// oaksLibrary/Regulatorer/fbSequenceController7Stages
// Pi-regulator 5-sekvens
{attribute 'initialize_on_call'}
FUNCTION_BLOCK fbSequenceController7Stages
VAR_INPUT
	bEnable : BOOL; // Aktiverar reglering
	rProcessValue : REAL; // Aktuellt Ärvärde 
	rSetpoint : REAL; // Aktuellt börvärde. Önskas separat kylbörvärde för kylsekvenser se inputen rCoolSetpoint.
	{attribute 'initialize_on_call'}
	rCoolSetpoint : REFERENCE TO REAL; //Om man önskar ha ett högre börvärde för kylsekvenser lägg denna här så väljs detta på de sekvenser där bActnSequenceX = TRUE. Lämnar man inputen tom körs rSetpoint på både kyl och värmesekvenser.
	rMinSeq1 : REAL := 0; 
	rMaxSeq1 : REAL := 100;
	bActnSequence1 : BOOL; // Gångriktning reglersekvens  (kylsekvens = TRUE)
	bBlockSequence1 : BOOL; // blockera denna sekvens kan användas exempelvis vid nattkyla
	rMinSeq2 : REAL := 0; 
	rMaxSeq2 : REAL := 100;
	bActnSequence2 : BOOL; // Gångriktning reglersekvens  (kylsekvens = TRUE)
	bBlockSequence2 : BOOL; // blockera denna sekvens kan användas exempelvis vid nattkyla
	rMinSeq3 : REAL := 0; 
	rMaxSeq3 : REAL := 100;
	bActnSequence3 : BOOL; // Gångriktning reglersekvens  (kylsekvens = TRUE)
	bBlockSequence3 : BOOL; // blockera denna sekvens kan användas exempelvis vid nattkyla
	rMinSeq4 : REAL := 0; 
	rMaxSeq4 : REAL := 100;
	bActnSequence4 : BOOL; // Gångriktning reglersekvens  (kylsekvens = TRUE)
	bBlockSequence4 : BOOL; // blockera denna sekvens kan användas exempelvis vid nattkyla
	rMinSeq5 : REAL := 0; 
	rMaxSeq5 : REAL := 100;
	bActnSequence5 : BOOL; // Gångriktning reglersekvens  (kylsekvens = TRUE)
	bBlockSequence5 : BOOL; // blockera denna sekvens kan användas exempelvis vid nattkyla
	rMinSeq6 : REAL := 0; 
	rMaxSeq6 : REAL := 100;
	bActnSequence6 : BOOL; // Gångriktning reglersekvens  (kylsekvens = TRUE)
	bBlockSequence6 : BOOL; // blockera denna sekvens kan användas exempelvis vid nattkyla
	rMinSeq7 : REAL := 0; 
	rMaxSeq7 : REAL := 100;
	bActnSequence7 : BOOL; // Gångriktning reglersekvens  (kylsekvens = TRUE)
	bBlockSequence7 : BOOL; // blockera denna sekvens kan användas exempelvis vid nattkyla
	rKpSequence1 : REAL; // Kp
	rKiSequence1 : UDINT; // Ki
	rDiSequence1 : UDINT; // D-tid (Derivata)
	rFDiSequence1 : UDINT; // Filter tid D (Derivata)
	rDzSequence1 : REAL :=0.1; //Dödzon
	rKpSequence2 : REAL; // Kp
	rKiSequence2 : UDINT; // Ki
	rDiSequence2 : UDINT; // D-tid (Derivata)
	rFDiSequence2 : UDINT; // Filter tid D (Derivata)
	rDzSequence2 : REAL :=0.1; //Dödzon
	rKpSequence3 : REAL; // Kp
	rKiSequence3 : UDINT; // Ki
	rDiSequence3 : UDINT; // D-tid (Derivata)
	rFDiSequence3 : UDINT; // Filter tid D (Derivata)
	rDzSequence3 : REAL :=0.1; //Dödzon
	rKpSequence4 : REAL; // Kp
	rKiSequence4 : UDINT; // Ki
	rDiSequence4 : UDINT; // D-tid (Derivata)
	rFDiSequence4 : UDINT; // Filter tid D (Derivata)
	rDzSequence4 : REAL :=0.1; //Dödzon
	rKpSequence5 : REAL; // Kp
	rKiSequence5 : UDINT; // Ki
	rDiSequence5 : UDINT; // D-tid (Derivata)
	rFDiSequence5 : UDINT; // Filter tid D (Derivata)
	rDzSequence5 : REAL :=0.1; //Dödzon
	rKpSequence6 : REAL; // Kp
	rKiSequence6 : UDINT; // Ki
	rDiSequence6 : UDINT; // D-tid (Derivata)
	rFDiSequence6 : UDINT; // Filter tid D (Derivata)
	rDzSequence6 : REAL :=0.1; //Dödzon
	rKpSequence7 : REAL; // Kp
	rKiSequence7 : UDINT; // Ki
	rDiSequence7 : UDINT; // D-tid (Derivata)
	rFDiSequence7 : UDINT; // Filter tid D (Derivata)
	rDzSequence7 : REAL :=0.1; //Dödzon
	iStartSequence : UDINT :=3; //Sekvens där regulator startar
	{attribute 'pingroup' := 'DeviationAlarm'}
	{attribute 'initialize_on_call'}
	rDevLimit : REFERENCE TO REAL := 0;
	{attribute 'pingroup' := 'DeviationAlarm'}
	bBlockHighAlarm : BOOL; // Blockera högtemplarm
	{attribute 'pingroup' := 'DeviationAlarm'}
	bBlockLowAlarm : BOOL; // Blockera lågtemplarm
	{attribute 'pingroup' := 'DeviationAlarm'}
	tAlarmDelay : TIME := T#5S; // larmfördröjning
END_VAR
VAR_OUTPUT
	rY : REAL; // Utsignal huvudregulator
	rOutputSequence1 : REAL;  // regulatorsignal
	rOutputSequence2 : REAL;  // regulatorsignal
	rOutputSequence3 : REAL;  // regulatorsignal
	rOutputSequence4 : REAL;  // regulatorsignal
	rOutputSequence5 : REAL;  // regulatorsignal
	rOutputSequence6 : REAL;  // regulatorsignal
	rOutputSequence7 : REAL;  // regulatorsignal
	{attribute 'pingroup' := 'DeviationAlarm'}
	bAlarmOutput : BOOL; //larmutgång
END_VAR
VAR
	rDevLimitInternal : REAL;
	fbDevAlarmPV: fbDevAlarm;
	rSetPointSequence1,rSetPointSequence2,rSetPointSequence3,rSetPointSequence4,rSetPointSequence5,rSetPointSequence6,rSetPointSequence7 : REAL; 	
	rTempMin,rTempMax : REAL; // tempvariabel för blockering av sekvenser 
	fbSeqLink01: Tc3_BA_Common.FB_BA_SeqLink;
	stSeqLink01 : Tc3_BA_Common.ST_BA_SeqLink;
	fbPidSeq: ARRAY[1..7] OF Tc3_BA_Common.FB_BA_SeqCtrl;
	iStartSequenceInternal : UDINT := 3;
END_VAR

	fbDevAlarmPV(
	tAlarmDelay:=tAlarmDelay , 
	bAutoReset:=TRUE , 
	bAlarmOutput=>bAlarmOutput , 
	bEnable:=bEnable AND mDevAlarmCheck() , 
	rProcessValue:=rProcessValue , 
	rSetPoint:=rSetpoint , 
	rDevLimit:=rDevLimitInternal , 
	bBlockHighAlarm:=bBlockHighAlarm , 
	bBlockLowAlarm:=bBlockLowAlarm );

	IF iStartSequence > 0 AND iStartSequence < 7 THEN
	 iStartSequenceInternal	 := 7 - iStartSequence;
	END_IF;
		
	
	fbSeqLink01(
	bEn:= bEnable, 
	udiSttCtrl:= iStartSequenceInternal, 
	udiIniSwiOvrDly_sec:= 5, 
	rX:= rProcessValue, 
	stSeqLink:=stSeqLink01 , 
	udiCurCtrl=> , 
	bSeqActv=> , 
	bNotRead=> , 
	bNoneOp=> , 
	udiRemTiIniSwiOvrDly_sec=> , 
	bErr=> , 
	sErrDescr=> );
		
	IF bBlockSequence1 THEN
		rTempMin := 0;
		rTempMax := 0;
	ELSE
		rTempMin := rMinSeq1;
		rTempMax := rMaxSeq1;
	END_IF
	rSetPointSequence1 := mCoolSetpointCheck(bActnSequence1);
	fbPidSeq[1](
	bEn:=bEnable , 
	rW:= rSetPointSequence1, 
	rX:=rProcessValue , 
	udiOpMode:= , 
	bActn:=bActnSequence1 , 
	rKp:= rKpSequence1, 
	udiTn_ms:=rKiSequence1*1000 , 
	udiTv_ms:=rDiSequence1*1000 , 
	udiTd_ms:=rFDiSequence1*1000 , 
	rYMax:=rTempMax , 
	rYMin:=rTempMin, 
	rNZ:= rDzSequence1, 
	udiCycCl:= , 
	bSync:= , 
	rSync:= , 
	rYSeqInit:= , 
	udiMyNum:= 7, 
	stSeqLink:=stSeqLink01 , 
	rY=> rOutputSequence1, 
	rE=> , 
	bErr=> , 
	sErrDescr=> );
	
	IF bBlockSequence2 THEN
		rTempMin := 0;
		rTempMax := 0;
	ELSE
		rTempMin := rMinSeq2;
		rTempMax := rMaxSeq2;
	END_IF
	rSetPointSequence2 := mCoolSetpointCheck(bActnSequence2);
	fbPidSeq[2](
	bEn:=bEnable , 
	rW:= rSetPointSequence2, 
	rX:= rProcessValue, 
	udiOpMode:= , 
	bActn:= bActnSequence2, 
	rKp:= rKpSequence2, 
	udiTn_ms:=rKiSequence2*1000 , 
	udiTv_ms:=rDiSequence2*1000 , 
	udiTd_ms:=rFDiSequence2*1000 , 
	rYMax:= rTempMax, 
	rYMin:=rTempMin , 
	rNZ:= rDzSequence2, 
	udiCycCl:= , 
	bSync:= , 
	rSync:= , 
	rYSeqInit:= , 
	udiMyNum:= 6, 
	stSeqLink:= stSeqLink01, 
	rY=> rOutputSequence2, 
	rE=> , 
	bErr=> , 
	sErrDescr=> );
	
	IF bBlockSequence3 THEN
		rTempMin := 0;
		rTempMax := 0;
	ELSE
		rTempMin := rMinSeq3;
		rTempMax := rMaxSeq3;
	END_IF
	rSetPointSequence3 := mCoolSetpointCheck(bActnSequence3);
	fbPidSeq[3](
	bEn:=bEnable , 
	rW:= rSetPointSequence3, 
	rX:= rProcessValue, 
	udiOpMode:= , 
	bActn:= bActnSequence3, 
	rKp:= rKpSequence3, 
	udiTn_ms:=rKiSequence3*1000 , 
	udiTv_ms:=rDiSequence3*1000 , 
	udiTd_ms:=rFDiSequence3*1000 , 
	rYMax:=rTempMax , 
	rYMin:= rTempMin, 
	rNZ:= rDzSequence3, 
	udiCycCl:= , 
	bSync:= , 
	rSync:= , 
	rYSeqInit:= , 
	udiMyNum:= 5, 
	stSeqLink:= stSeqLink01, 
	rY=> rOutputSequence3, 
	rE=> , 
	bErr=> , 
	sErrDescr=> );
	
	IF bBlockSequence4 THEN
		rTempMin := 0;
		rTempMax := 0;
	ELSE
		rTempMin := rMinSeq4;
		rTempMax := rMaxSeq4;
	END_IF
	rSetPointSequence4 := mCoolSetpointCheck(bActnSequence4);
	fbPidSeq[4](
	bEn:=bEnable , 
	rW:= rSetPointSequence4, 
	rX:= rProcessValue, 
	udiOpMode:= , 
	bActn:= bActnSequence4, 
	rKp:= rKpSequence4, 
	udiTn_ms:=rKiSequence4*1000 , 
	udiTv_ms:=rDiSequence4*1000 , 
	udiTd_ms:=rFDiSequence4*1000 , 
	rYMax:=rTempMax , 
	rYMin:= rTempMin, 
	rNZ:= rDzSequence4, 
	udiCycCl:= , 
	bSync:= , 
	rSync:= , 
	rYSeqInit:= , 
	udiMyNum:= 4, 
	stSeqLink:= stSeqLink01, 
	rY=> rOutputSequence4, 
	rE=> , 
	bErr=> , 
	sErrDescr=> );
	
	IF bBlockSequence5 THEN
		rTempMin := 0;
		rTempMax := 0;
	ELSE
		rTempMin := rMinSeq5;
		rTempMax := rMaxSeq5;
	END_IF
	rSetPointSequence5 := mCoolSetpointCheck(bActnSequence5);
	fbPidSeq[5](
	bEn:=bEnable , 
	rW:= rSetPointSequence5, 
	rX:= rProcessValue, 
	udiOpMode:= , 
	bActn:= bActnSequence5, 
	rKp:= rKpSequence5, 
	udiTn_ms:=rKiSequence5*1000 , 
	udiTv_ms:=rDiSequence5*1000 , 
	udiTd_ms:=rFDiSequence5*1000 , 
	rYMax:=rTempMax , 
	rYMin:= rTempMin, 
	rNZ:= rDzSequence5, 
	udiCycCl:= , 
	bSync:= , 
	rSync:= , 
	rYSeqInit:= , 
	udiMyNum:= 3, 
	stSeqLink:= stSeqLink01, 
	rY=> rOutputSequence5, 
	rE=> , 
	bErr=> , 
	sErrDescr=> );
	
	IF bBlockSequence6 THEN
		rTempMin := 0;
		rTempMax := 0;
	ELSE
		rTempMin := rMinSeq6;
		rTempMax := rMaxSeq6;
	END_IF
	rSetPointSequence6 := mCoolSetpointCheck(bActnSequence6);
	fbPidSeq[6](
	bEn:=bEnable , 
	rW:= rSetPointSequence6, 
	rX:= rProcessValue, 
	udiOpMode:= , 
	bActn:= bActnSequence6, 
	rKp:= rKpSequence6, 
	udiTn_ms:=rKiSequence6*1000 , 
	udiTv_ms:=rDiSequence6*1000 , 
	udiTd_ms:=rFDiSequence6*1000 , 
	rYMax:=rTempMax , 
	rYMin:= rTempMin, 
	rNZ:= rDzSequence6, 
	udiCycCl:= , 
	bSync:= , 
	rSync:= , 
	rYSeqInit:= , 
	udiMyNum:= 2, 
	stSeqLink:= stSeqLink01, 
	rY=> rOutputSequence6, 
	rE=> , 
	bErr=> , 
	sErrDescr=> );
	
	IF bBlockSequence7 THEN
		rTempMin := 0;
		rTempMax := 0;
	ELSE
		rTempMin := rMinSeq7;
		rTempMax := rMaxSeq7;
	END_IF
	rSetPointSequence7 := mCoolSetpointCheck(bActnSequence7);
	fbPidSeq[7](
	bEn:=bEnable , 
	rW:= rSetPointSequence7, 
	rX:= rProcessValue, 
	udiOpMode:= , 
	bActn:= bActnSequence7, 
	rKp:= rKpSequence7, 
	udiTn_ms:=rKiSequence7*1000 , 
	udiTv_ms:=rDiSequence7*1000 , 
	udiTd_ms:=rFDiSequence7*1000 , 
	rYMax:=rTempMax , 
	rYMin:= rTempMin, 
	rNZ:= rDzSequence7, 
	udiCycCl:= , 
	bSync:= , 
	rSync:= , 
	rYSeqInit:= , 
	udiMyNum:= 1, 
	stSeqLink:= stSeqLink01, 
	rY=> rOutputSequence7, 
	rE=> , 
	bErr=> , 
	sErrDescr=> );

// Publik metod för att kolla ifall det finns någon kylsekvens i regleringen. Kan exempelvis användas för att blockera högavvikelselarm vid hög utetemperatur då kylsekvens saknas.
METHOD PUBLIC mContainsCoolingSequence : BOOL
mContainsCoolingSequence := bActnSequence1 OR bActnSequence2 OR bActnSequence3 OR bActnSequence4 OR bActnSequence5;
END_METHOD

// Metod för att kolla ifall det är en kylsekvens och om det i sådant fall är något knutet på rCoolSetpoint
METHOD PRIVATE mCoolSetpointCheck : REAL // Valt börvärde
VAR_INPUT
	bActn : BOOL; // Koll av gångriktning
END_VAR
IF NOT bActn THEN
	mCoolSetpointCheck := rSetpoint;
ELSE
	IF __ISVALIDREF(rCoolSetpoint) THEN 
		mCoolSetpointCheck := rCoolSetpoint;
	ELSE
		mCoolSetpointCheck := rSetpoint;
	END_IF
END_IF
END_METHOD

// Kolla ifall något är knutet på inputen rDevLimit. Är inget knutet där inaktiveras avvikelselarmet.
METHOD PRIVATE mDevAlarmCheck : BOOL // Valt börvärde
IF __ISVALIDREF(rDevLimit) THEN 
	mDevAlarmCheck := TRUE;
	rDevLimitInternal := rDevLimit;
ELSE
	mDevAlarmCheck := FALSE;
END_IF
END_METHOD

END_FUNCTION_BLOCK

// oaksLibrary/Skicka värden mellan plc/Inbyggda taggar/fbReadAdsBoolGeneralWp
// Läser önskat real-värde från annan PLC enligt Oaks-standard
// Robert H, 2021-11-23
// Testat 2021-11-23
FUNCTION_BLOCK fbReadAdsBoolGeneralWp
VAR_INPUT
	Enable			: BOOL := TRUE;					// Start
	AmsNetId    	: T_AmsNetId; 					// AMS Net ID till enhet som skall avläsas
    AdsPort     	: T_AmsPort := 851; 			// ADS-port till enhet som skall avläsas
	AdsTimeout    	: TIME := DEFAULT_ADS_TIMEOUT; 	// ADS-timeout
	SymbolName  	: T_MaxString; 					// Symbol-/variabelnamn för den variabel som skall avläsas. Hela sökväg skall anges tex. LA1.GP11.PV
	Interval		: TIME := T#10S;				// Önskat intervall för läsning
	ErrDelay		: TIME := T#5S;					// Larmfördröjning för fel
	FallbackVal		: BOOL;					// Värde vid kom.fel eller manuellt val av fallback (knyt t ex lokal utegivare om den finns)
	UseFallback		: BOOL;							// Sätts om fallbackvärde ska användas automatiskt vid fel
	ForceFallback	: BOOL;							// Sätts om fallbackvärde ska användas ovillkorligt
	Apparatskap 	: STRING := 'ASXX'; 			// Skriv här vilket apparatskåp utetemperaturen tas emot från. Endast för visning i PV4-tagg.
END_VAR
VAR_OUTPUT
	{attribute 'OPC.UA.DA' := '1'}
	Output 			: BOOL; 	//Utetemperatur hämtat från apparatskåp via ADS
	{attribute 'OPC.UA.DA' := '1'}
	FAULT AT %M* 	: BOOL; 	//Kommunikationsfel mottagning av värde via ADS~wp:
	{attribute 'OPC.UA.DA' := '1'}
	PV8 AT %M* 		: STRING;  	//Inställt amsNetId och apparatskåp~wp:
END_VAR
VAR	
	fbReadVal	: fbReadADSBool;
END_VAR

IF Enable THEN
	fbReadVal(enable := Enable, amsNetId := amsNetId, adsPort := adsPort, adsTimeout := adsTimeout, symbolName := SymbolName, interval := interval, errDelay := errDelay, fallbackVal := fallbackVal, useFallback := UseFallback, forceFallback := forceFallback);
	
	Output	:= fbReadVal.bOutputVar;							// Skriv avläst värde					
	PV8		:= CONCAT(amsNetId, CONCAT('-', Apparatskap));		// Bygg ihop ID-sträng för visning
	FAULT	:= fbReadVal.bErr;									// Sätt fellarm
END_IF;

END_FUNCTION_BLOCK

// oaksLibrary/Skicka värden mellan plc/fbReadADSBool
// Läser önskad bool-variabel från annan ADS-enhet
// Robert H, 2021-11-23
// Testat 2021-11-23
FUNCTION_BLOCK fbReadADSBool
VAR_INPUT
    amsNetId    	: T_AmsNetId; 					//AMS Net ID till enhet som skall avläsas
    adsPort     	: T_AmsPort := 851; 			// ADS-port till den enhet som skall avlä
	symbolName  	: T_MaxString; 					// Symbol-/variabelnamn för den variabel som skall avläsas. Hela sökväg skall anges tex. LA1.GP11.PV
	enable			: BOOL;							// Start
	adsTimeout    	: TIME := DEFAULT_ADS_TIMEOUT; 	// ADS-timout
	interval		: TIME := T#10S;				// Önskat intervall för läsning
	errDelay		: TIME := T#5S;					// Larmfördröjning för fel
	fallbackVal		: BOOL := FALSE;				// Värde vid kom.fel eller manuellt val av fallback
	useFallback		: BOOL := FALSE;				// Sätts om fallbackvärde får användas vid fel
	forceFallback	: BOOL := FALSE;				// Sätts om fallbackvärde ska användas ovillkorligt 			
END_VAR
VAR_OUTPUT
	bBusy     	: BOOL; 			// Upptagen
	bErr     	: BOOL; 			// Fel (via Err-flagga från funktioner, eller om case landat i error state över 10 ggr)
	nErrId    	: UDINT;			// Felkod
	SymInfo  	: SYMINFOSTRUCT; 	// Datastruktur avläst symbolinfo
	bOutputVar	: BOOL;				// Avläst värde
END_VAR
VAR
    errInternal   		: BOOL; 					// Fel
	fbErrorTon 			: TON;  					// Tillslagsfördröjning felindikering
	fbErrorTof 			: TOF;						// Frånslagsfördröjning felindikering
	fbReadSymInfoByName	: PLC_ReadSymInfoByName;	// Maska ut symboladress
 	fbAdsRead			: ADSREAD;					// ADS-block 
	state 				: INT;						// Case-index
	CycleTimer			: TON;						// Intervalltimer för ADS-funktioner
	outputValInternal	: BOOL;						// Avläst värde internt
	StErrCnt			: INT;						// Antal gånger i rad case landat i error state
END_VAR

// Från/tillslagsfördröjning kom.fel
fbErrorTof(IN := , PT := interval + T#5S , Q => errInternal);
fbErrorTon(IN := errInternal OR (amsNetId = '') OR (StErrCnt > 10), PT := errDelay);

bErr := fbErrorTon.Q OR amsNetId = '';

CycleTimer(IN := state = 0 AND (NOT bBusy), PT := Interval);	// Intervalltimer för ADS-funktioner

CASE state OF
	0:
		IF CycleTimer.Q AND enable THEN
			bBusy := TRUE;
			fbErrorTof.IN := FALSE;			
			state := 1;
		END_IF	
	
	1: // Read symbol info by specified name
					
			bBusy := TRUE;
			fbErrorTof.IN := FALSE;
					
			fbReadSymInfoByName(
			NETID:= amsNetId, 
			PORT:= adsPort, 
			SYMNAME:= symbolName, 
			START:= TRUE, 
			TMOUT:= adsTimeout, 
			BUSY=> bBusy, 
			ERR=> fbErrorTof.IN, 
			ERRID=> nErrId, 
			SYMINFO=> SymInfo);
			
			IF NOT bBusy THEN
				IF NOT errInternal AND SymInfo.symDataType = 'BOOL' THEN
					fbReadSymInfoByName( Start := FALSE );
					 state := 2; // Success / Goto next
				ELSE
					fbReadSymInfoByName( Start := FALSE );
					state := 100; // Error
				END_IF
			END_IF
		
	2: // Read symbol value
			
			fbAdsRead(
			NETID:= amsNetId, 
			PORT:= adsPort, 
			IDXGRP:= syminfo.idxGroup, 
			IDXOFFS:= syminfo.idxOffset, 
			LEN:= SIZEOF(outputValInternal), 
			DESTADDR:= ADR(outputValInternal), 
			READ:= TRUE, 
			TMOUT:= adsTimeout, 
			BUSY=> bBusy, 
			ERR=> fbErrorTof.IN, 
			ERRID=> nErrId);
									
			IF NOT bBusy THEN
				IF NOT errInternal THEN
					fbAdsRead( READ := FALSE );
					state := 0; // Success / Goto next
					StErrCnt := 0;
				ELSE
					fbAdsRead( READ := FALSE );
					state := 100; // Error
				END_IF
			END_IF
	
	100: // Error handling
	StErrCnt := StErrCnt + 1;	
	state := 0;
END_CASE

IF (bErr AND useFallback) OR forceFallback THEN
	bOutputVar := fallbackVal;
ELSIF bErr THEN
	bOutputVar := FALSE;
ELSE
	bOutputVar := outputValInternal;
END_IF

END_FUNCTION_BLOCK

// oaksLibrary/Skicka värden mellan plc/Inbyggda taggar/fbReadAdsRealGeneralWp
// Läser önskat real-värde från annan PLC enligt Oaks-standard
// Robert H, 2021-11-23
// Testat 2021-11-23
FUNCTION_BLOCK fbReadAdsRealGeneralWp
VAR_INPUT
	Enable			: BOOL := TRUE;					// Start
	AmsNetId    	: T_AmsNetId; 					// AMS Net ID till enhet som skall avläsas
    AdsPort     	: T_AmsPort := 851; 			// ADS-port till enhet som skall avläsas
	AdsTimeout    	: TIME := DEFAULT_ADS_TIMEOUT; 	// ADS-timeout
	SymbolName  	: T_MaxString; 					// Symbol-/variabelnamn för den variabel som skall avläsas. Hela sökväg skall anges tex. LA1.GP11.PV
	Interval		: TIME := T#10S;				// Önskat intervall för läsning
	ErrDelay		: TIME := T#5S;					// Larmfördröjning för fel
	FallbackVal		: REAL := 0.0;					// Värde vid kom.fel eller manuellt val av fallback (knyt t ex lokal utegivare om den finns)
	UseFallback		: BOOL;							// Sätts om fallbackvärde ska användas automatiskt vid fel
	ForceFallback	: BOOL;							// Sätts om fallbackvärde ska användas ovillkorligt
	Apparatskap 	: STRING := 'ASXX'; 			// Skriv här vilket apparatskåp utetemperaturen tas emot från. Endast för visning i PV4-tagg.
END_VAR
VAR_OUTPUT
	{attribute 'OPC.UA.DA' := '1'}
	Output 			: REAL; 	//Värde hämtat från apparatskåp via ADS (Knyts till egenskapad tagg)
	{attribute 'OPC.UA.DA' := '1'}
	FAULT AT %M* 	: BOOL; 	//Kommunikationsfel mottagning av värde via ADS~wp:
	{attribute 'OPC.UA.DA' := '1'}
	PV8 AT %M* 		: STRING;  	//Inställt amsNetId och apparatskåp~wp:
END_VAR
VAR	
	fbReadVal	: fbReadADSReal;
END_VAR

IF Enable THEN
	fbReadVal(enable := Enable, amsNetId := amsNetId, adsPort := adsPort, adsTimeout := adsTimeout, symbolName := SymbolName, interval := interval, errDelay := errDelay, fallbackVal := fallbackVal, useFallback := UseFallback, forceFallback := forceFallback);
	
	Output	:= fbReadVal.rOutputVar;							// Skriv avläst värde					
	PV8		:= CONCAT(amsNetId, CONCAT('-', Apparatskap));		// Bygg ihop ID-sträng för visning
	FAULT	:= fbReadVal.bErr;									// Sätt fellarm
END_IF;

END_FUNCTION_BLOCK

// oaksLibrary/Skicka värden mellan plc/fbReadADSReal
// Läser önskad real-variabel från annan ADS-enhet
// Robert H, 2021-11-23
// Testat 2021-11-23
FUNCTION_BLOCK fbReadADSReal
VAR_INPUT
    amsNetId    	: T_AmsNetId; 					//AMS Net ID till enhet som skall avläsas
    adsPort     	: T_AmsPort := 851; 			// ADS-port till den enhet som skall avlä
	symbolName  	: T_MaxString; 					// Symbol-/variabelnamn för den variabel som skall avläsas. Hela sökväg skall anges tex. LA1.GP11.PV
	enable			: BOOL;							// Start
	adsTimeout    	: TIME := DEFAULT_ADS_TIMEOUT; 	// ADS-timout
	interval		: TIME := T#10S;				// Önskat intervall för läsning
	errDelay		: TIME := T#5S;					// Larmfördröjning för fel
	fallbackVal		: REAL := 0.0;					// Värde vid kom.fel eller manuellt val av fallback
	useFallback		: BOOL := FALSE;				// Sätts om fallbackvärde får användas vid fel
	forceFallback	: BOOL := FALSE;				// Sätts om fallbackvärde ska användas ovillkorligt 			
END_VAR
VAR_OUTPUT
	bBusy     	: BOOL; 			// Upptagen
	bErr     	: BOOL; 			// Fel (via Err-flagga från funktioner, eller om case landat i error state över 10 ggr)
	nErrId    	: UDINT;			// Felkod
	SymInfo  	: SYMINFOSTRUCT; 	// Datastruktur avläst symbolinfo
	rOutputVar	: REAL;				// Avläst värde
END_VAR
VAR
    errInternal   		: BOOL; 					// Fel
	fbErrorTon 			: TON;  					// Tillslagsfördröjning felindikering
	fbErrorTof 			: TOF;						// Frånslagsfördröjning felindikering
	fbReadSymInfoByName	: PLC_ReadSymInfoByName;	// Maska ut symboladress
 	fbAdsRead			: ADSREAD;					// ADS-block 
	state 				: INT;						// Case-index
	CycleTimer			: TON;						// Intervalltimer för ADS-funktioner
	outputValInternal	: REAL;						// Avläst värde internt
	StErrCnt			: INT;						// Antal gånger i rad case landat i error state
END_VAR

// Från/tillslagsfördröjning kom.fel
fbErrorTof(IN := , PT := interval + T#5S , Q => errInternal);
fbErrorTon(IN := errInternal OR (amsNetId = '') OR (StErrCnt > 10), PT := errDelay);

bErr := fbErrorTon.Q OR amsNetId = '';

CycleTimer(IN := state = 0 AND (NOT bBusy), PT := Interval);	// Intervalltimer för ADS-funktioner

CASE state OF
	0:
		IF CycleTimer.Q AND enable THEN
			bBusy := TRUE;
			fbErrorTof.IN := FALSE;			
			state := 1;
		END_IF	
	
	1: // Read symbol info by specified name
					
			bBusy := TRUE;
			fbErrorTof.IN := FALSE;
					
			fbReadSymInfoByName(
			NETID:= amsNetId, 
			PORT:= adsPort, 
			SYMNAME:= symbolName, 
			START:= TRUE, 
			TMOUT:= adsTimeout, 
			BUSY=> bBusy, 
			ERR=> fbErrorTof.IN, 
			ERRID=> nErrId, 
			SYMINFO=> SymInfo);
			
			IF NOT bBusy THEN
				IF NOT errInternal AND SymInfo.symDataType = 'REAL' THEN
					fbReadSymInfoByName( Start := FALSE );
					 state := 2; // Success / Goto next
				ELSE
					fbReadSymInfoByName( Start := FALSE );
					state := 100; // Error
				END_IF
			END_IF
		
	2: // Read symbol value
	
			fbAdsRead(
			NETID:= amsNetId, 
			PORT:= adsPort, 
			IDXGRP:= syminfo.idxGroup, 
			IDXOFFS:= syminfo.idxOffset, 
			LEN:= SIZEOF(outputValInternal), 
			DESTADDR:= ADR(outputValInternal), 
			READ:= TRUE, 
			TMOUT:= adsTimeout, 
			BUSY=> bBusy, 
			ERR=> fbErrorTof.IN, 
			ERRID=> nErrId);
									
			IF NOT bBusy THEN
				IF NOT errInternal THEN
					fbAdsRead( READ := FALSE );
					state := 0; // Success / Goto next
					StErrCnt := 0;
				ELSE
					fbAdsRead( READ := FALSE );
					state := 100; // Error
				END_IF
			END_IF
	
	100: // Error handling
		StErrCnt := StErrCnt + 1;
		state := 0;
END_CASE

IF (bErr AND useFallback) OR forceFallback THEN
	rOutputVar := fallbackVal;
ELSIF bErr THEN
	rOutputVar := 0.0;
ELSE
	rOutputVar := outputValInternal;
END_IF

END_FUNCTION_BLOCK

// oaksLibrary/Skicka värden mellan plc/Inbyggda taggar/fbReadAdsRealOutdoorMeantempWp
// Läser momentan och medelvärde utetemp från annan PLC enligt oaks-standard
// Robert H, 2021-11-23
// Testat 2021-11-23
FUNCTION_BLOCK fbReadAdsRealOutdoorMeantempWp
VAR_INPUT
	Enable			: BOOL := TRUE;					// Start
	AmsNetId    	: T_AmsNetId; 					// AMS Net ID till enhet som skall avläsas
	sApparatskap 	: STRING 	:= 'ASXX'; 			// Skriv här vilket apparatskåp utetemperaturen tas emot från. Endast för visning i PV4-tagg.
    AdsPort     	: T_AmsPort := 851; 			// ADS-port till den enhet som skall avläsas
	AdsTimeout    	: TIME := DEFAULT_ADS_TIMEOUT; 	// ADS-timout
	Interval		: TIME := T#10S;				// Önskat intervall för läsning
	ErrDelay		: TIME := T#5S;					// Larmfördröjning för fel
	UseFallback		: BOOL;							// Sätts om fallbackvärde ska användas automatiskt vid fel
	FallbackVal		: REAL := 0.0;					// Värde vid kom.fel eller manuellt val av fallback (knyt t ex lokal utegivare om den finns)
	ForceFallback	: BOOL;							// Sätts om fallbackvärde ska användas ovillkorligt
END_VAR
VAR_OUTPUT
	{attribute 'OPC.UA.DA' := '1'}
	PV  AT %M* : REAL; //Utetemperatur hämtat från apparatskåp via ads.~wp:[unit]°C[format]0.0
	{attribute 'OPC.UA.DA' := '1'}
	PV1  AT %M* : REAL; //Utetemperatur medel hämtat från apparatskåp via ads.~wp:[unit]°C[format]0.0
	{attribute 'OPC.UA.DA' := '1'}
	FAULT AT %M* : BOOL; //Kommunikationsfel mottagning utetemperatur~wp:
	{attribute 'OPC.UA.DA' := '1'}
	PV4 AT %M* : STRING;   //Inställt amsNetId och apparatskåp~wp:
END_VAR
VAR	
	fbUtetempMom	: fbReadADSReal;
	fbUtetempMed	: fbReadADSReal;
END_VAR

IF enable THEN
	fbUtetempMom(Enable := enable, amsNetId := amsNetId, adsPort := adsPort, adsTimeout := adsTimeout, symbolName := 'oaksGVL.rOutdoorTemp', interval := interval, errDelay := errDelay, fallbackVal := fallbackVal, useFallback := UseFallback, forceFallback := forceFallback);
	oaksGVL.rOutdoorTemp := fbUtetempMom.rOutputVar;
	
	fbUtetempMed(Enable := enable, amsNetId := amsNetId, adsPort := adsPort, adsTimeout := adsTimeout, symbolName := 'oaksGVL.rOutdoorTempMean', interval := interval, errDelay := errDelay, fallbackVal := fallbackVal, useFallback := UseFallback, forceFallback := forceFallback);
	oaksGVL.rOutdoorTempMean := fbUtetempMed.rOutputVar;
	
	PV		:= oaksGVL.rOutdoorTemp;							// Skriv utetemp till utvariabel	
	PV1		:= oaksGVL.rOutdoorTempMean;						// Skriv utetemp medel till utvariabel				
	PV4		:= CONCAT(amsNetId, CONCAT('-', sApparatskap));		// Bygg ihop ID-sträng för visning
	FAULT	:= fbUtetempMom.bErr OR fbUtetempMed.bErr;			// Sätt fel
END_IF;

END_FUNCTION_BLOCK

// oaksLibrary/Skicka värden mellan plc/Inbyggda taggar/fbReadAdsRealOutdoortempWp
// Läser utetemp från annan PLC enligt oaks-standard
// Robert H, 2021-11-23
// Testat 2021-11-23
FUNCTION_BLOCK fbReadAdsRealOutdoortempWp
VAR_INPUT
	Enable			: BOOL := TRUE;					// Start
	AmsNetId    	: T_AmsNetId; 					// AMS Net ID till enhet som skall avläsas
	sApparatskap 	: STRING 	:= 'ASXX'; 			// Skriv här vilket apparatskåp utetemperaturen tas emot från. Endast för visning i PV4-tagg.
    AdsPort     	: T_AmsPort := 851; 			// ADS-port till den enhet som skall avläsas
	AdsTimeout    	: TIME := DEFAULT_ADS_TIMEOUT; 	// ADS-timout
	Interval		: TIME := T#10S;				// Önskat intervall för läsning
	ErrDelay		: TIME := T#5S;					// Larmfördröjning för fel
	UseFallback		: BOOL;							// Sätts om fallbackvärde ska användas automatiskt vid fel
	FallbackVal		: REAL := 0.0;					// Värde vid kom.fel eller manuellt val av fallback (knyt t ex lokal utegivare om den finns)
	ForceFallback	: BOOL;							// Sätts om fallbackvärde ska användas ovillkorligt
END_VAR
VAR_OUTPUT
	{attribute 'OPC.UA.DA' := '1'}
	PV  AT %M* : REAL; //Utetemperatur hämtat från apparatskåp via ads.~wp:[unit]°C[format]0.0
	{attribute 'OPC.UA.DA' := '1'}
	FAULT AT %M* : BOOL; //Kommunikationsfel mottagning utetemperatur~wp:
	{attribute 'OPC.UA.DA' := '1'}
	PV4 AT %M* : STRING;   //Inställt amsNetId och apparatskåp~wp:
END_VAR
VAR	
	fbUtetempMom	: fbReadADSReal;
	fbUtetempMed	: fbReadADSReal;
END_VAR

IF enable THEN
	fbUtetempMom(Enable := enable, amsNetId := amsNetId, adsPort := adsPort, adsTimeout := adsTimeout, symbolName := 'oaksGVL.rOutdoorTemp', interval := interval, errDelay := errDelay, fallbackVal := fallbackVal, useFallback := UseFallback, forceFallback := forceFallback);
	oaksGVL.rOutdoorTemp := fbUtetempMom.rOutputVar;
	
	PV		:= oaksGVL.rOutdoorTemp;							// Skriv utetemp till utvariabel					
	PV4		:= CONCAT(amsNetId, CONCAT('-', sApparatskap));		// Bygg ihop ID-sträng för visning
	FAULT	:= fbUtetempMom.bErr OR fbUtetempMed.bErr;			// Sätt fel
END_IF;

END_FUNCTION_BLOCK

// oaksLibrary/Skicka värden mellan plc/Inbyggda taggar/fbReadAdsTempSensorWp
// Läser tempgivare från annan PLC enligt oaks-standard
// Robert H, 2021-11-23
// Testat 2021-11-23
FUNCTION_BLOCK fbReadAdsTempSensorWp
VAR_INPUT
	Enable			: BOOL := TRUE;					// Start
	AmsNetId    	: T_AmsNetId; 					// AMS Net ID till enhet som skall avläsas
    AdsPort     	: T_AmsPort := 851; 			// ADS-port till enhet som skall avläsas
	AdsTimeout    	: TIME := DEFAULT_ADS_TIMEOUT; 	// ADS-timeout
	SymbolName  	: T_MaxString; 					// Symbol-/variabelnamn för den variabel som skall avläsas. Hela sökväg skall anges tex. LA1.GT11.PV
	Interval		: TIME := T#10S;				// Önskat intervall för läsning
	ErrDelay		: TIME := T#5S;					// Larmfördröjning för fel
	FallbackVal		: REAL := 0.0;					// Värde vid kom.fel eller manuellt val av fallback (knyt t ex lokal utegivare om den finns)
	UseFallback		: BOOL;							// Sätts om fallbackvärde ska användas automatiskt vid fel
	ForceFallback	: BOOL;							// Sätts om fallbackvärde ska användas ovillkorligt
	Apparatskap 	: STRING := 'ASXX'; 			// Skriv här vilket apparatskåp utetemperaturen tas emot från. Endast för visning i PV4-tagg.
END_VAR
VAR_OUTPUT
	{attribute 'OPC.UA.DA' := '1'}
	PV AT %M*		: REAL; 	//Temperatur~wp:[unit]°C[format]0.0[trendoptions]i:300
	{attribute 'OPC.UA.DA' := '1'}
	FAULT AT %M* 	: BOOL; 	//Kommunikationsfel mottagning av värde via ADS~wp:
	{attribute 'OPC.UA.DA' := '1'}
	PV8 AT %M* 		: STRING;  	//Inställt amsNetId och apparatskåp~wp:
END_VAR
VAR	
	fbReadVal	: fbReadADSReal;
END_VAR

IF Enable THEN
	fbReadVal(enable := Enable, amsNetId := amsNetId, adsPort := adsPort, adsTimeout := adsTimeout, symbolName := SymbolName, interval := interval, errDelay := errDelay, fallbackVal := fallbackVal, useFallback := UseFallback, forceFallback := forceFallback);
	
	PV		:= fbReadVal.rOutputVar;							// Skriv avläst värde					
	PV8		:= CONCAT(amsNetId, CONCAT('-', Apparatskap));		// Bygg ihop ID-sträng för visning
	FAULT	:= fbReadVal.bErr;									// Sätt fellarm
END_IF;

END_FUNCTION_BLOCK

// oaksLibrary/Skicka värden mellan plc/fbReadAdsInt
// Läser önskad int-variabel från annan ADS-enhet
// Robert H, 2021-11-23
// Testat 2021-11-23
FUNCTION_BLOCK fbReadAdsInt
VAR_INPUT
    amsNetId    	: T_AmsNetId; 					//AMS Net ID till enhet som skall avläsas
    adsPort     	: T_AmsPort := 851; 			// ADS-port till den enhet som skall avlä
	symbolName  	: T_MaxString; 					// Symbol-/variabelnamn för den variabel som skall avläsas. Hela sökväg skall anges tex. LA1.GP11.PV
	enable			: BOOL;							// Start
	adsTimeout    	: TIME := DEFAULT_ADS_TIMEOUT; 	// ADS-timout
	interval		: TIME := T#10S;				// Önskat intervall för läsning
	errDelay		: TIME := T#5S;					// Larmfördröjning för fel
	fallbackVal		: INT := 0;					// Värde vid kom.fel eller manuellt val av fallback
	useFallback		: BOOL := FALSE;				// Sätts om fallbackvärde får användas vid fel
	forceFallback	: BOOL := FALSE;				// Sätts om fallbackvärde ska användas ovillkorligt 			
END_VAR
VAR_OUTPUT
	bBusy     	: BOOL; 			// Upptagen
	bErr     	: BOOL; 			// Fel (via Err-flagga från funktioner, eller om case landat i error state över 10 ggr)
	nErrId    	: UDINT;			// Felkod
	SymInfo  	: SYMINFOSTRUCT; 	// Datastruktur avläst symbolinfo
	iOutputVar	: INT;				// Avläst värde
END_VAR
VAR
    errInternal   		: BOOL; 					// Fel
	fbErrorTon 			: TON;  					// Tillslagsfördröjning felindikering
	fbErrorTof 			: TOF;						// Frånslagsfördröjning felindikering
	fbReadSymInfoByName	: PLC_ReadSymInfoByName;	// Maska ut symboladress
 	fbAdsRead			: ADSREAD;					// ADS-block 
	state 				: INT;						// Case-index
	CycleTimer			: TON;						// Intervalltimer för ADS-funktioner
	outputValInternal	: INT;						// Avläst värde internt
	StErrCnt			: INT;						// Antal gånger i rad case landat i error state
END_VAR

// Från/tillslagsfördröjning kom.fel
fbErrorTof(IN := , PT := interval + T#5S, Q => errInternal);
fbErrorTon(IN := errInternal OR (amsNetId = '') OR (StErrCnt > 10), PT := errDelay);

bErr := fbErrorTon.Q OR amsNetId = '';

CycleTimer(IN := state = 0 AND (NOT bBusy), PT := Interval);	// Intervalltimer för ADS-funktioner

CASE state OF
	0:
		IF CycleTimer.Q AND enable THEN
			bBusy := TRUE;
			fbErrorTof.IN := FALSE;			
			state := 1;
		END_IF	
	
	1: // Read symbol info by specified name
					
			bBusy := TRUE;
			fbErrorTof.IN := FALSE;
						
			fbReadSymInfoByName(
			NETID:= amsNetId, 
			PORT:= adsPort, 
			SYMNAME:= symbolName, 
			START:= TRUE, 
			TMOUT:= adsTimeout, 
			BUSY=> bBusy, 
			ERR=> fbErrorTof.IN, 
			ERRID=> nErrId, 
			SYMINFO=> SymInfo);
			
			IF NOT bBusy THEN
				IF NOT errInternal AND SymInfo.symDataType = 'INT' THEN
					fbReadSymInfoByName( Start := FALSE );
					 state := 2; // Success / Goto next
				ELSE
					fbReadSymInfoByName( Start := FALSE );
					state := 100; // Error
				END_IF
			END_IF
		
	2: // Read symbol value
	
			fbAdsRead(
			NETID:= amsNetId, 
			PORT:= adsPort, 
			IDXGRP:= syminfo.idxGroup, 
			IDXOFFS:= syminfo.idxOffset, 
			LEN:= SIZEOF(outputValInternal), 
			DESTADDR:= ADR(outputValInternal), 
			READ:= TRUE, 
			TMOUT:= adsTimeout, 
			BUSY=> bBusy, 
			ERR=> fbErrorTof.IN, 
			ERRID=> nErrId);
									
			IF NOT bBusy THEN
				IF NOT errInternal THEN
					fbAdsRead( READ := FALSE );
					state := 0; // Success / Goto next
					StErrCnt := 0;
				ELSE
					fbAdsRead( READ := FALSE );
					state := 100; // Error
				END_IF
			END_IF
	
	100: // Error handling
		StErrCnt := StErrCnt + 1;
		state := 0;
END_CASE

IF (bErr AND useFallback) OR forceFallback THEN
	iOutputVar := fallbackVal;
ELSIF bErr THEN
	iOutputVar := 0;
ELSE
	iOutputVar := outputValInternal;
END_IF

END_FUNCTION_BLOCK

// oaksLibrary/Skicka värden mellan plc/fbReadAdsRealOutdoortemp
// Används för att ta emot utetemp. Skriver internt i blocket till oaksgvl.rOutdoorTemp
FUNCTION_BLOCK fbReadAdsRealOutdoortemp
VAR_INPUT
    amsNetId    : T_AmsNetId; //AMS Net ID till enhet som skall avläsas
    adsPort     : T_AmsPort := 851; // ADS-port till den enhet som skall avläsas
  	symbolName  : T_MaxString := 'oaksgvl.rOutdoorTemp'; // Symbol-/variabelnamn för den variabel som skall avläsas. Hela sökväg skall anges tex. LA1.GP11.PV
    enable    : BOOL; // Start
    adsTimeout    : TIME := DEFAULT_ADS_TIMEOUT; // ADS-timout
	bTestMode : BOOL; // Aktivera denna input för att inaktivera skrivning till oaksgvl.rOutdoorTemp
END_VAR
VAR_OUTPUT
    bBusy     : BOOL; //Upptagen
    bErr     : BOOL; // Fel
    nErrId    : UDINT; // Fel-kod
    SymInfo  : SYMINFOSTRUCT; // Datastruktur avläst symbolinfo
	rOutputVar : REAL; // Avläst värde
END_VAR
VAR
    bErrInternal      : BOOL; // Fel
	fbErrorTon : TON;
	fbErrorTof : TOF;
//Get symbol info
	fbReadSymInfoByName: PLC_ReadSymInfoByName;
 	fbAdsRead: ADSREAD; 
	nState : INT;
END_VAR

IF NOT bTestMode THEN
	IF NOT bErr THEN
		oaksgvl.rOutdoorTemp := rOutputVar;
	ELSE
		oaksgvl.rOutdoorTemp := 0.0;
	END_IF
END_IF;

fbErrorTof(IN:= , PT:=T#5S , Q=>bErrInternal , ET=> );
fbErrorTon(IN:=bErrInternal OR amsNetId = '' , PT:=T#10S , Q=>bErr , ET=> );
CASE nState OF
    0:
        IF enable THEN
            bBusy := TRUE;
            fbErrorTof.IN := FALSE;			
			nState := 1;
		END_IF	
	
	1: // Read symbol info by specified name
					
			bBusy := TRUE;
            fbErrorTof.IN := FALSE;

			fbReadSymInfoByName(
			NETID:= amsNetId, 
			PORT:= adsPort, 
			SYMNAME:= symbolName, 
			START:= TRUE, 
			TMOUT:= adsTimeout, 
			BUSY=> bBusy, 
			ERR=> fbErrorTof.IN, 
			ERRID=> nErrId, 
			SYMINFO=> SymInfo);
            
			IF NOT bBusy THEN
            	IF NOT bErrInternal AND SymInfo.symDataType = 'REAL' THEN
               		fbReadSymInfoByName( Start := FALSE );
					 nState := 2; // Success / Goto next
            	ELSE
                	fbReadSymInfoByName( Start := FALSE );
					nState := 100; // Error
            	END_IF
       		END_IF
        
	2: // Read symbol value

			fbAdsRead(
			NETID:= amsNetId, 
			PORT:= adsPort, 
			IDXGRP:= syminfo.idxGroup, 
			IDXOFFS:= syminfo.idxOffset, 
			LEN:= SIZEOF(rOutputVar), 
			DESTADDR:= ADR(rOutputVar), 
			READ:= TRUE, 
			TMOUT:= adsTimeout, 
			BUSY=> bBusy, 
			ERR=> fbErrorTof.IN, 
			ERRID=> nErrId);
									
			IF NOT bBusy THEN
            	IF NOT bErrInternal THEN
            	    fbAdsRead( READ := FALSE );
					nState := 0; // Success / Goto next
            	ELSE
                	fbAdsRead( READ := FALSE );
					nState := 100; // Error
            	END_IF
       		END_IF
	
	
    100: // Error handling
        nState := 0;
END_CASE

END_FUNCTION_BLOCK

// oaksLibrary/System/fbBK9050
//Oaks AB 2020-06-10
//Funktionsblock för övervakning av bus-fel/kommunikationsfel med 
FUNCTION_BLOCK fbBK9050
VAR_INPUT
	
END_VAR
VAR_OUTPUT
	//Interna fel buss-kopplare
	{attribute 'OPC.UA.DA' := '1'}
	AL AT %M* : BOOL; //IO-fel~wp:
	{attribute 'OPC.UA.DA' := '1'}
	PV1 AT %M* : STRING; //Fel~wp:
	//Almänna fel buss-kopplare
	{attribute 'OPC.UA.DA' := '1'}
	AL1 AT %M* : BOOL; //Kommunikationsfel~wp:
	{attribute 'OPC.UA.DA' := '1'}
	PV2 AT %M* : STRING; //Fel~wp:
	
END_VAR
VAR	
	couplerStateIn AT %I*: UINT; //Ingång från BK9050/Inputs/CouplerState
	boxStateIn AT %I*: UINT; //Ingång från BK9050/Inputs/BoxState
END_VAR

//Interna fel buss-kopplare
IF couplerStateIn <> 0 THEN
	AL := TRUE;
ELSE
	AL := FALSE;
END_IF

CASE couplerStateIn OF
	0: PV1 := 'Inget fel';
	1: PV1 := 'Bus-terminal fel';
	2: PV1 := 'Konfigurationsfel';
	
END_CASE

//Almänna fel buss-kopplare
IF boxStateIn <> 0 THEN
	AL1 := TRUE;
ELSE
	AL1 := FALSE;
END_IF

CASE boxStateIn OF
	0: PV2 := 'Inget fel';
	1: PV2 := 'Inga ingångar mottagna';
	2: PV2 := 'Utgångar avaktiverade';
	4: PV2 := 'Ingen kommunikation';
	8: PV2 := 'Gamla ingångar';
	16: PV2 := 'Ogiltlig ingångs längd';
	32: PV2 := 'Ogiltlig utgångs längd';
	
END_CASE

END_FUNCTION_BLOCK

// oaksLibrary/System/fbOaksSystem
// Funktionsblock för systemhantering av PLC
FUNCTION_BLOCK fbOaksSystem
VAR_INPUT
	tSekvensstartTid1 : TIME := T#5S; //Sekvensstart 1 tid
	tSekvensstartTid2 : TIME := T#10S; //Sekvensstart 2 tid
	tSekvensstartTid3 : TIME := T#15S; //Sekvensstart 3 tid
	tSekvensstartTid4 : TIME := T#20S; //Sekvensstart 4 tid
	tSekvensstartTid5 : TIME := T#25S; //Sekvensstart 5 tid
	tSekvensstartTid6 : TIME := T#30S; //Sekvensstart 6 tid
	tSekvensstartTid7 : TIME := T#35S; //Sekvensstart 7 tid
	tSekvensstartTid8 : TIME := T#40S; //Sekvensstart 8 tid
	tSekvensstartTid9 : TIME := T#45S; //Sekvensstart 9 tid
	tSekvensstartTid10 : TIME := T#50S; //Sekvensstart 10 tid
	tSekvensstartTid11 : TIME := T#60S; //Sekvensstart 11 tid
	tSekvensstartTid12 : TIME := T#65S; //Sekvensstart 12 tid
	tSekvensstartTid13 : TIME := T#70S; //Sekvensstart 13 tid
	tSekvensstartTid14 : TIME := T#75S; //Sekvensstart 14 tid
	tSekvensstartTid15 : TIME := T#80S; //Sekvensstart 15 tid
	
	M AT %M* : BOOL; //Manuell reset av larm beräkningsfel~wp:[trendoptions]i:14400, t:1
END_VAR

VAR_OUTPUT
	{attribute 'OPC.UA.DA' := '1'}
	AL AT %M* : BOOL; //Kritiskt beräkningsfel i PLC (kontakta OAKS)~wp:[alarmoptions]p:1
	{attribute 'OPC.UA.DA' := '1'}
	FAULT AT %M* : BOOL; //Fel på KBUS-system (kontakta OAKS)~wp:[alarmoptions]p:1
	{attribute 'OPC.UA.DA' := '1'}
	AL8 AT %M* : BOOL; //Okänd plc-modell~wp:[alarmoptions]p:3
	{attribute 'OPC.UA.DA' := '1'}
	PV8 AT %M* : STRING; //Plc-modell~wp:
	{attribute 'OPC.UA.DA' := '1'}
	PV 		: INT; // År~wp:
	{attribute 'OPC.UA.DA' := '1'}
	PV1 	: INT; // Månad(1-12)~wp:
	{attribute 'OPC.UA.DA' := '1'}
	PV2 	: INT; // Dag (1-31)~wp:
	{attribute 'OPC.UA.DA' := '1'}
	PV3		: INT; // Veckodag (1-7)~wp:
	{attribute 'OPC.UA.DA' := '1'}
	PV4 	: INT; // Timme (0-23)~wp:
	{attribute 'OPC.UA.DA' := '1'}
	PV5 	: INT; // Minut (0-59)~wp:
	{attribute 'OPC.UA.DA' := '1'}
	PV6 	: INT; // Sekund (0-59)~wp:
	{attribute 'OPC.UA.DA' := '1'}
	PV7 AT %M* : STRING; //Datum och tid från plc~wp:
	{attribute 'OPC.UA.DA' := '1'}
	PV9 AT %M* : STRING; //Orsak FAULT (KBUS)~wp:
	bRTCFault : BOOL;	//Fel i realtidsklocka (RTC-batteri slut samt ingen NTP-konfiguration)
END_VAR

VAR
	bInit : BOOL := FALSE;	//För uppstartsfunktioner
	
	fbHardwareModelInfo01 : fbHardwareModelInfo;
	fbAlarmfbHardwareModelInfo: fbAlarm;
	
	fbPLC_SystemTime: Tc3_BA.FB_BA_GetTime;
	stTime		: tc2_ba.TIMESTRUCT;
	FB_BA_GetTime01 : tc2_ba.FB_BA_GetTime; 
	FB_BA_ExtTiSt01 : tc2_ba.FB_BA_ExtTiSt;	
	uiInitCyCnt : UINT := 0;	
	
	fbS_UPS_CX5130				: FB_S_UPS_CX51x0;
	fbS_UPS_CX8190				: FB_S_UPS_CX81xx;
	fbS_UPS_CX9020				: FB_S_UPS_CX9020_U900;
	
	fbR_TrigPowerFailure		: Tc2_Standard.R_TRIG;
	fbCountPowerFailure			: Tc2_Standard.CTU;
	bResetCounterPowerFailures	: BOOL; // If TRUE the fbCountPowerFailure is reset to 0
	fbR_ResetCounter			: Tc2_Standard.R_TRIG;	
	bBootDataLoaded				: BOOL; // If TRUE bootdata file loaded. Normal behaviour.
	bOldBootDataLoaded			: BOOL; // IF TRUE old bootdata file is loaded. bootdata-file missing or corrupt.

	fbTonSekvensstart1  : TON; //Sekvensstart 1  global variabel sätts till true efter inställd tid
	fbTonSekvensstart2  : TON; //Sekvensstart 2  global variabel sätts till true efter inställd tid
	fbTonSekvensstart3  : TON; //Sekvensstart 3  global variabel sätts till true efter inställd tid
	fbTonSekvensstart4  : TON; //Sekvensstart 4  global variabel sätts till true efter inställd tid
	fbTonSekvensstart5  : TON; //Sekvensstart 5  global variabel sätts till true efter inställd tid
	fbTonSekvensstart6  : TON; //Sekvensstart 6  global variabel sätts till true efter inställd tid
	fbTonSekvensstart7  : TON; //Sekvensstart 7  global variabel sätts till true efter inställd tid
	fbTonSekvensstart8  : TON; //Sekvensstart 8  global variabel sätts till true efter inställd tid
	fbTonSekvensstart9  : TON; //Sekvensstart 9  global variabel sätts till true efter inställd tid
	fbTonSekvensstart10 : TON; //Sekvensstart 10 global variabel sätts till true efter inställd tid
	fbTonSekvensstart11 : TON; //Sekvensstart 11 global variabel sätts till true efter inställd tid
	fbTonSekvensstart12 : TON; //Sekvensstart 12 global variabel sätts till true efter inställd tid
	fbTonSekvensstart13 : TON; //Sekvensstart 13 global variabel sätts till true efter inställd tid
	fbTonSekvensstart14 : TON; //Sekvensstart 14 global variabel sätts till true efter inställd tid
	fbTonSekvensstart15 : TON; //Sekvensstart 15 global variabel sätts till true efter inställd tid

	fbPLC_WritePersistentData: Tc3_BA.FB_BA_WrtPersistDat;
	fbTimerWritePersistent: TON;
	bManualTrigg		: BOOL;	 // Manual trigger for writing persistent data
	fbRTrigManual: Tc2_Standard.R_TRIG;
	fbRTrigExecuted: Tc2_Standard.R_TRIG;

	fbKBUSInitTON 				: TON;				//Init-timer 
	nKbusState AT%I*			: UINT; 			//State for actual CX-BK. Linked to actual CX-BK.
	bKbusFailure				: BOOL; 			//IF TRUE KBUS-failure is active
	fbDeviceReset				: IOF_DeviceReset; 	//Functionblock för reset of KBUS. The hardcoded DEVICEID on FB must match the ID of the CX-BK
	bResetKbus					: BOOL;				//Internal variable for 
	fbRisingEdgeKbus			: R_TRIG;			//Autoreset		
	nRetriggIterator 			: INT 	:= 0;		//Counts up if the Kbusreset failed
	fbRetrigTimeOut 			: TON;				//Timer återstart
	bManualResetKBUS 			: BOOL 	:=FALSE;	//Manual Kbusreset. Is used when bResetKBUSAutomatically is to FALSE or the max number of Kbusreset retries is counted.
	fbRisingEdgeKbusManReset	: R_TRIG;			//Man. reset
	bKbusErrorMaxRestarted		: BOOL;				//Indicates that the limit of trying to reset Kbus is reached 
	bResetKbusInt				: BOOL;				//KBUS reset
	bKbusStateNotLinked			: BOOL;				//KBUS State ej länkad till IO-enhet
	nKbusResetCnt				: BYTE := 0;		//Räknare för felsökning
	bKBusInit					: BOOL := FALSE;	//KBUS init-flagga
	fbKbusAlarm 				: fbAlarm;			//KBUS larmblock				

	fbCheck1					: fbEdge;
	fbCheck2					: fbEdge;
	fbCheck3					: fbEdge;
	fbCheck4					: fbEdge;
	fbCheck5					: fbEdge;
	fbCheck6					: fbEdge;
	fbCheck7					: fbEdge;
	fbCheck8					: fbEdge;
	fbCheck9					: fbEdge;
	fbCheck10					: fbEdge;
	fbImplicitCheckAlarm		: fbAlarm;
END_VAR

VAR PERSISTENT
	dtTimeLastPowerFailure		: DT;		// Last Time Power Failure
	nNumberOfPowerFailures		: UDINT;	// Number of Power Failures since last reset of counter
	
	bActivate			: BOOL	:=TRUE;		// If TRUE cyclic writing of persistent data according to 
	nCycleTime			: TIME	:=T#24H; 	// The time cycle for writing of persistent data
	dtLastTimeExecuted	: DT	;			// Last time executed writing of persistent data
	
	bResetKBUSAutomatically 	: BOOL	:= TRUE;	//TRUE=Automatic reset of KbusFailure, FALSE=Manual reset of Kbusfailure
	tRetrigTime 				: TIME 	:= T#30S;	//How often Kbusreset is reactivated if the last attempt is not succesfully 
	nMaxRetries					: INT	:= 60;		//How many retries if the automatic reset is not succesful.
END_VAR

//Sekvensstart
	fbTonSekvensstart1(IN:=TRUE , PT:=tSekvensstartTid1 , Q=>oaksgvl.bSekvensstart1 , ET=> );
	fbTonSekvensstart2(IN:=TRUE , PT:=tSekvensstartTid2 , Q=>oaksgvl.bSekvensstart2 , ET=> );
	fbTonSekvensstart3(IN:=TRUE , PT:=tSekvensstartTid3 , Q=>oaksgvl.bSekvensstart3 , ET=> );
	fbTonSekvensstart4(IN:=TRUE , PT:=tSekvensstartTid4 , Q=>oaksgvl.bSekvensstart4 , ET=> );
	fbTonSekvensstart5(IN:=TRUE , PT:=tSekvensstartTid5 , Q=>oaksgvl.bSekvensstart5 , ET=> );
	fbTonSekvensstart6(IN:=TRUE , PT:=tSekvensstartTid6 , Q=>oaksgvl.bSekvensstart6 , ET=> );
	fbTonSekvensstart7(IN:=TRUE , PT:=tSekvensstartTid7 , Q=>oaksgvl.bSekvensstart7 , ET=> );
	fbTonSekvensstart8(IN:=TRUE , PT:=tSekvensstartTid8 , Q=>oaksgvl.bSekvensstart8 , ET=> );
	fbTonSekvensstart9(IN:=TRUE , PT:=tSekvensstartTid9 , Q=>oaksgvl.bSekvensstart9 , ET=> );
	fbTonSekvensstart10(IN:=TRUE , PT:=tSekvensstartTid10 , Q=>oaksgvl.bSekvensstart10 , ET=> );
	fbTonSekvensstart11(IN:=TRUE , PT:=tSekvensstartTid11 , Q=>oaksgvl.bSekvensstart11 , ET=> );
	fbTonSekvensstart12(IN:=TRUE , PT:=tSekvensstartTid12 , Q=>oaksgvl.bSekvensstart12 , ET=> );
	fbTonSekvensstart13(IN:=TRUE , PT:=tSekvensstartTid13 , Q=>oaksgvl.bSekvensstart13 , ET=> );
	fbTonSekvensstart14(IN:=TRUE , PT:=tSekvensstartTid14 , Q=>oaksgvl.bSekvensstart14 , ET=> );
	fbTonSekvensstart15(IN:=TRUE , PT:=tSekvensstartTid15 , Q=>oaksgvl.bSekvensstart15 , ET=> );
//Slut


//Konfigurering av passiva givar-kort
	oaksGVL.fbPassiveAnalogInConfigTonReset(IN:=oaksgvl.bPassiveAnalogInConfig , PT:=T#30S , Q=> , ET=> );
	IF oaksGVL.fbPassiveAnalogInConfigTonReset.Q THEN
		oaksgvl.bPassiveAnalogInConfig := FALSE;
	END_IF
//Slut


//Realtidsklocka
	FB_BA_GetTime01(bEn :=TRUE);	
	stTime := FB_BA_GetTime01.stSysTi;
	
	IF uiInitCyCnt < 10 THEN	//Sätt larm för fel i realtidsklocka om inläst år är <2023 efter 10 cykler
		uiInitCyCnt := uiInitCyCnt + 1;
	ELSE
		bRTCFault := stTime.wYear < 2023;
	END_IF
	
	PV 	:=WORD_TO_INT (stTime.wYear); 
	oaksGVL.iYear := PV;
	PV1 :=WORD_TO_INT (stTime.wMonth);
	oaksGVL.iMonth := PV1;
	PV2 :=WORD_TO_INT (stTime.wDay);
	oaksGVL.iDay := PV2;

	//Beckhoffs "veckodag" går 0-6, denna säkerställer att det är enligt beskrivningstext för PV3 taggen
	//Tidiger = PV3 :=WORD_TO_INT (stTime.wDayOfWeek);
	CASE WORD_TO_INT (stTime.wDayOfWeek) OF
		0: PV3:= 7;
		1: PV3:= 1;
		2: PV3:= 2;
		3: PV3:= 3;
		4: PV3:= 4;
		5: PV3:= 5;
		6: PV3:= 6;
	END_CASE
	oaksGVL.iDayOfWeek := PV3;
	
	PV4 :=WORD_TO_INT (stTime.wHour);
	oaksGVL.iHour := PV4;
	PV5 :=WORD_TO_INT (stTime.wMinute);
	oaksGVL.iMinute := PV5;
	PV6 :=WORD_TO_INT (stTime.wSecond);
	oaksGVL.iSecond := PV6;
	
	oaksGVL.iHourAndMinute := (oaksGVL.iHour *100) + oaksGVL.iMinute;
	
	PV7 := CONCAT(CONCAT(CONCAT(CONCAT(CONCAT(CONCAT(CONCAT(CONCAT(CONCAT(CONCAT(INT_TO_STRING(PV),'-'),INT_TO_STRING(PV1)),'-'),INT_TO_STRING(PV2)), ' '), INT_TO_STRING(PV4)),':'),INT_TO_STRING(PV5)),':'),INT_TO_STRING(PV6));
	
	//SystemTime (används av andra funktioner)
	fbPLC_SystemTime( bEn:= TRUE, sNetId:= , udiUpdRtc_sec:= , bUpdRtc:= , bRdySysTi=> , bRdyTiZoInfo=> , bRdyRTC=> , udiRemTiUpd_sec=> , stSysTi=> , stUTC=> , dtSysTi=> , dtUTC=> , udiCurrentTime_ms=> , eTiZId=> , bErr=> , sErrDescr=> );
//Slut


//Kontrollera PLC-modell, sätt larm om okänd (dvs ej stöd av Oaks)
	fbHardwareModelInfo01(strHardwareModel=> );
	
	PV8 := fbHardwareModelInfo01.strHardwareModel;
	fbAlarmfbHardwareModelInfo(bInput := 	fbHardwareModelInfo01.strHardwareModel <> 'CX8190' AND 
											fbHardwareModelInfo01.strHardwareModel <> 'CX5110-0115' AND
											fbHardwareModelInfo01.strHardwareModel <> 'CX5130-0155' AND
											fbHardwareModelInfo01.strHardwareModel <> 'CX5130-0175' AND
											fbHardwareModelInfo01.strHardwareModel <> 'CX9020-B000', 
											tAlarmDelay:=T#10S, 
											bAutoReset:=, 
											bAlarmOutput=>AL8 );
//Slut										


//Hantering av 1-sek UPS & skrivning av persistent data
	IF fbHardwareModelInfo01.strHardwareModel = 'CX8190' THEN
		fbS_UPS_CX8190(
		sNetID:= , 
		iPLCPort:= , 
		tTimeout:= , 
		eUpsMode:= , 
		ePersistentMode:= , 
		tRecoverTime:= , 
		bPowerFailDetect=> , 
		eState=> );
		fbR_TrigPowerFailure( CLK := fbS_UPS_CX8190.bPowerFailDetect, Q=> );
	ELSIF LEFT(fbHardwareModelInfo01.strHardwareModel, 4) = 'CX51'  THEN //Hela CX5100-serien
		fbS_UPS_CX5130(
		sNetID:= , 
		iPLCPort:= , 
		iUPSPort:= , 
		tTimeout:= , 
		eUpsMode:= , 
		ePersistentMode:= , 
		tRecoverTime:= , 
		bPowerFailDetect=> , 
		eState=> );	
		fbR_TrigPowerFailure( CLK := fbS_UPS_CX5130.bPowerFailDetect, Q=> );
	ELSIF fbHardwareModelInfo01.strHardwareModel = 'CX9020-B000' THEN
		fbS_UPS_CX9020(
		sNetID:= , 
		iPLCPort:= , 
		tTimeout:= , 
		eUpsMode:= , 
		ePersistentMode:= , 
		tRecoverTime:= , 
		bPowerFailDetect=> , 
		eState=> );
		fbR_TrigPowerFailure( CLK := fbS_UPS_CX9020.bPowerFailDetect, Q=> );
	END_IF
	
	IF fbR_TrigPowerFailure.Q THEN
		dtTimeLastPowerFailure := fbPLC_SystemTime.dtSysTi;
		nNumberOfPowerFailures := nNumberOfPowerFailures +1;
	END_IF
	
	fbR_ResetCounter( CLK := bResetCounterPowerFailures , Q=> );
	
	IF fbR_ResetCounter.Q THEN
		nNumberOfPowerFailures := 0;
		bResetCounterPowerFailures := FALSE;
	END_IF
	
	//Write Persistent Data
	fbTimerWritePersistent( IN := bActivate AND NOT fbTimerWritePersistent.Q, PT:=nCycleTime, Q=> , ET=> );
	
	fbRTrigManual( CLK := bManualTrigg, Q=> );
	
	IF fbRTrigManual.Q THEN bManualTrigg := FALSE; END_IF
	
	fbPLC_WritePersistentData( bStt:= fbTimerWritePersistent.Q OR fbRTrigManual.Q, udiInitSttDly_sec:= , bBusy=> , udiRemTiInitSttDly_sec=> , bErr=> , sErrDescr=> );
	
	fbRTrigExecuted( CLK := fbPLC_WritePersistentData.bBusy, Q=> );
	
	IF fbRTrigExecuted.Q THEN dtLastTimeExecuted := fbPLC_SystemTime.dtSysTi; END_IF;
//Slut

	
//KBUS-hantering
	IF NOT bInit OR NOT fbKBUSInitTON.Q THEN	//Sätt bitar i state-flagga vid uppstart (ej bit 0)
		nKbusState := 254;
		fbKBUSInitTON(IN := TRUE, PT := T#10S);
	ELSE
		bKbusStateNotLinked := nKbusState = 254;	//Sätt felflagga för ej linkad Kbus-enhet om kbus-state ej förändrats från uppstart.
		bKbusFailure := nKbusState.0;				//Sätt felflagga för Kbus-fel om bit 0 i state är aktiv
		
		fbRisingEdgeKbus(CLK:= (bResetKBUSAutomatically AND (bKbusFailure OR fbDeviceReset.ERR)), Q=> );	//Trigga reset vid kBus-fel eller misslyckad device reset
		fbRisingEdgeKbusManReset(CLK:= bManualResetKBUS, Q=> );												//Manuell reset
		
		IF fbRisingEdgeKbusManReset.Q THEN bManualResetKBUS := FALSE; END_IF	//Återställ man.reset
		
		IF fbRisingEdgeKbusManReset.Q OR fbRisingEdgeKbus.Q THEN	//Starta reset
			bResetKbus := TRUE;
			bResetKbusInt := TRUE;
			bKbusErrorMaxRestarted := FALSE;
			nRetriggIterator := 0;
			nKbusResetCnt := nKbusResetCnt + 1;	
		END_IF
		
		//Initiera deviceID till reset-funktion (oklar lösning, bör ersättas med säker metod)
		IF fbHardwareModelInfo01.strHardwareModel = 'CX8190' OR fbHardwareModelInfo01.strHardwareModel = 'CX9020-B000' OR fbHardwareModelInfo01.strHardwareModel = 'CX5110-0115' THEN
			fbDeviceReset.DEVICEID := 2;
		ELSIF fbHardwareModelInfo01.strHardwareModel = 'CX5130-0155' OR fbHardwareModelInfo01.strHardwareModel = 'CX5130-0175' THEN
			fbDeviceReset.DEVICEID := 3;
		END_IF
		
		//Kör devicereset vid kommando samt initerad buss
		fbDeviceReset(
			NETID:= , 
			RESET:= bResetKbusInt AND bKBusInit, 
			TMOUT:= T#3S, 
			BUSY=> , 
			ERR=> , 
			ERRID=> );
			
		IF fbDeviceReset.BUSY THEN bResetKbusInt := FALSE; END_IF	//Återställ internflagga
		
		//Återstart av reset enligt timerintervall, med max antal återstarter
		fbRetrigTimeOut(IN:= (NOT fbDeviceReset.BUSY AND bResetKbus AND (bKbusFailure OR fbDeviceReset.ERR) AND nRetriggIterator <= nMaxRetries), PT:= tRetrigTime, Q=> , ET=> );
		
		IF fbRetrigTimeOut.Q THEN
			nRetriggIterator := nRetriggIterator +1;
			bResetKbusInt := TRUE;
		END_IF
		
		//Larm vid max antal återställningsförsök eller om state-variabel ej länkad eller om fel från kbus reset-block
		fbKbusAlarm(bInput:= (nRetriggIterator > 5) OR bKbusStateNotLinked OR fbDeviceReset.ERR, tAlarmDelay:= T#5S, bAutoReset:=TRUE , bAlarmOutput=> FAULT);	
		
		//Sätt flagga för max återställning samt återställ reset
		IF nRetriggIterator > nMaxRetries THEN bKbusErrorMaxRestarted := TRUE; END_IF
		IF bKbusErrorMaxRestarted OR NOT (bKbusFailure OR fbDeviceReset.ERR) THEN bResetKbus := FALSE; END_IF
		
		//Skriv felorsak till strängvariabel
		IF bKbusStateNotLinked THEN
			PV9 := 'nKbusState ej länkad';
		ELSIF fbDeviceReset.ERR THEN
			PV9 := 'KBUS reset misslyckad';
		ELSIF bKbusFailure THEN
			PV9 := 'Fel i busskopplare';
		ELSE
			PV9 := 'Inget fel';
		END_IF
		
		//Kör en manual reset och sätt kbus init första programvarv
		IF NOT bKBusInit THEN bManualResetKBUS := TRUE; END_IF; 
		bKBusInit := TRUE;
		
	END_IF
//Slut


//Hantering av larm för Implicit-kontroller (allvarligt beräkningsfel i PLC)
	fbCheck1(anyInput := oaksGVL.udiCheckBounds, bIncr := TRUE);
	fbCheck2(anyInput := oaksGVL.udiCheckDivDInt, bIncr := TRUE);
	fbCheck3(anyInput := oaksGVL.udiCheckDivLInt, bIncr := TRUE);
	fbCheck4(anyInput := oaksGVL.udiCheckDivLReal, bIncr := TRUE);
	fbCheck5(anyInput := oaksGVL.udiCheckDivReal, bIncr := TRUE);
	fbCheck6(anyInput := oaksGVL.udiCheckLRangeSigned, bIncr := TRUE);
	fbCheck7(anyInput := oaksGVL.udiCheckLRangeUnsigned, bIncr := TRUE);
	fbCheck8(anyInput := oaksGVL.udiCheckPointer, bIncr := TRUE);
	fbCheck9(anyInput := oaksGVL.udiCheckRangeSigned, bIncr := TRUE);
	fbCheck10(anyInput := oaksGVL.udiCheckRangeUnsigned, bIncr := TRUE);
	
	fbImplicitCheckAlarm.bInput := 	fbCheck1.bEdgeF OR fbCheck2.bEdgeF OR fbCheck3.bEdgeF OR fbCheck4.bEdgeF OR fbCheck5.bEdgeF OR 
									fbCheck6.bEdgeF OR fbCheck7.bEdgeF OR fbCheck8.bEdgeF OR fbCheck9.bEdgeF OR fbCheck10.bEdgeF;
									
	fbImplicitCheckAlarm(bAutoReset := M, tAlarmDelay := T#0S, bAlarmOutput => AL);
	M := FALSE;
//Slut


bInit := TRUE;	//Sätt bInit för andra funktioner

END_FUNCTION_BLOCK

// oaksLibrary/System/fbSumAlarmWp
// Används detta block vid behov av att köra summalarm filtrerat på klassning
// Använd sedan nedanstående script i webport. Körs som loopande lämpligtvis med 10 sekunders intervall.
(*
	var alarms = getActiveAlarmList(true);
	var iLarmlampa = 0;
	// Skriv in dina parametrar här nedan
	var sWatchdogTagg = "AS01_SUMMALARMSLAMPA_A_PV8";
	var sSummaLarmsLampaTagg = "AS01_SUMMALARMSLAMPA_A_V";
	var sNamnPaEnhet = "AS01";
	var sPrioritet = "1"; 
	
	if (tagRead(sWatchdogTagg) == 1) // Växlande toggling larmlampa tänds i plc om denna inte togglar
	{
		tags[sWatchdogTagg].WriteValue(0, true);
	}
	else
	{
		tags[sWatchdogTagg].WriteValue(1, true);
	}
	for (var i=0;i<alarms.Count;i++) { // Kollar om det finns något aktivt larm i angiven enhet med angiven larmklassning
	  if(tags[alarms[i].Tag].Device.Name == sNamnPaEnhet && tags[alarms[i].Tag].AlarmOptions.Priority == sPrioritet && (alarms[i].State == Moldeo.WebPortCommon.AlarmStates.ALARM_NACK || alarms[i].State == Moldeo.WebPortCommon.AlarmStates.ALARM)) {
			iLarmlampa = 1;
	  }  
	} 
	tags[sSummaLarmsLampaTagg].WriteValue(iLarmlampa, true);
*)

FUNCTION_BLOCK fbSumAlarmWp
VAR_INPUT
END_VAR
VAR_OUTPUT
	{attribute 'OPC.UA.DA' := '1'}
	CMD AT %Q*  : BOOL;//Summalarmslamapa~wp:[format]0[trendoptions]i:14400, t:1
	{attribute 'OPC.UA.DA' := '1'}
	FAULT AT %M*  : BOOL;//Watchdog summalarmslampa apparatskåp. Script för summalarm ur funktion~wp:[format]0
END_VAR
VAR
	{attribute 'OPC.UA.DA' := '1'}
	V AT %M*  : BOOL;//Summalarmstagg sätts från webport~wp:[format]0[trendoptions]i:14400, t:1
	{attribute 'OPC.UA.DA' := '1'}
	PV8 AT %M*  : BOOL;//Watchdog-tagg. Summalarmslampa går till om denna inte togglar efter en minut~wp:[format]0
	
	timer01 : ton;
	timer02 : ton;
	fbAlarm: fbAlarm;
END_VAR

//Watchdog summalarmslampa apparatskåp. Script för summalarm ur funktion
timer01(IN:= NOT PV8, PT:=T#60S , Q=> , ET=> );
timer02(IN:= PV8, PT:=T#60S , Q=> , ET=> );
fbAlarm(bInput:= timer01.Q OR timer02.Q, tAlarmDelay:= T#1S, bAutoReset:= TRUE, bAlarmOutput=>FAULT);


// Sätter summalarmslampa
CMD := V OR FAULT;

END_FUNCTION_BLOCK

// oaksLibrary/Utsignal DO_AO/Motorer/fbGenericMotorHeatCool
// Generic "Motorblock" för digital utsignal med driftsvar/summalarm med möjlighet att handställa utsignal. Larmar vid handställning eller utebliven driftindikering/summalarm.
// Inbyggda taggar (start, stop, fördröjning) för webport. Ingång bModeHeat används för att växla mellan startvillkor värme och kyla.
// Utetemp från oaksGVL används ifall ingen annan givare kopplas till ingång rTempToUse.
FUNCTION_BLOCK fbGenericMotorHeatCool
VAR_INPUT
	rTempToUse : ANY; //Temperatur för start/stopp. Om inget kopplas används oaksGVL.rOutdoorTemp
	bModeHeat : BOOL := TRUE; //Alternativ för start/stopptemperaturer. TRUE = Startar när temperaturen understiger startgräns, stoppar när temperaturen överstiger stoppgräns. FALSE = Cool = tvärtom.
	bServiceStop : BOOL; //Serviceomkopplare. Utgång går från om denna ingång är till
	bSafe: BOOL; //Säkerhetsvillkor - Blockerar utsignal i autoläge samt blockerar handställning. Måste vara TRUE för att block ska kunna köras. 
	bPumpmotionConfig : BOOL; //TRUE = global funktion för pumpmotion används. Kräver att bSafe är till för att pumpmotion ska kunna köras. Kräver att ett block av typen fbPumpmotion deklareras och körs.
	bSumAlarmConfig	: BOOL; //TRUE = summalarm FALSE = driftindikering
	bInputInvert :BOOL; //Invertering av digtal insignal
	bAutoReset : BOOL := TRUE; //Auto-reset utav driftfel
	bHandsetBlock : BOOL; //Används för blockering av handställning utan att blockera utsignal i autoläge. OBS! - För säkerhetsvillkor se ingång bSafe!
	tAlarmDelay : TIME := T#3S; //Larmfördröjning	
END_VAR
VAR_OUTPUT
	{attribute 'OPC.UA.DA' := '1'}
	CMD AT %Q*  : BOOL; //Utsignal~wp:[trendoptions]i:14400, t:1
	{attribute 'OPC.UA.DA' := '1'}
	V 	AT %M* 	: BOOL; //Driftindikering~wp:[trendoptions]i:14400, t:1
	{attribute 'OPC.UA.DA' := '1'}
	AL 	AT %M*	: BOOL; //Driftfel~wp:[alarmoptions]p:2
	{attribute 'OPC.UA.DA' := '1'}
	AL8 AT %M* 	: BOOL; //Utsignal handställd~wp:[alarmoptions]p:3
	{attribute 'OPC.UA.DA' := '1'}
	PV7 AT %M* 	: UDINT; //Drifttid~wp:[unit]timmar[format]0[trendoptions]i:300
	{attribute 'OPC.UA.DA' := '1'}
	PV8 AT %M* 	: STRING; //Konfiguration startvillkor & digital ingång~wp:
END_VAR
VAR
	bStart : BOOL; // Startvillkor
	{attribute 'OPC.UA.DA' := '1'}
	RST AT %M* : BOOL := FALSE; //Nollställ drifttid~wp:[trendoptions]i:14400, t:1
	tStartDelay : TIME := T#1S; //Startfördröjning
	rTempUsed : REAL;
	bInternalStart : BOOL;
	bIndication AT %I* : BOOL; //Om bSumAlarmConfig = TRUE summalarmsingång annars driftindikering.
	bProcessedIndication :BOOL; 
	bAlarm : BOOL;
	fbAlarm1, fbAlarm2 : fbAlarm;
	bPumpMotionStart : BOOL; //Starta pumpmotion
	fbStartDelay: TON; // Startfördröjning
	fbStopDelay : TOF; // Stoppfördröjning
	fbOperatingHours_1: fbOperatingHours;
	bIntStart: BOOL;
END_VAR
VAR_INPUT PERSISTENT
	{attribute 'OPC.UA.DA' := '1'}
	M AT %M* : BOOL; //Handställning~wp:[trendoptions]i:14400, t:1
	{attribute 'OPC.UA.DA' := '1'}
	MCMD AT %M* : BOOL; //Styrsignal handställning~wp:[trendoptions]i:14400, t:1
	{attribute 'OPC.UA.DA' := '1'}
	SP3 AT %M* : INT := 15; //Stoppfördröjning~wp:[unit]min
	{attribute 'OPC.UA.DA' := '1'}
	SP2 AT %M* : REAL := 12; //Gränsvärde stopp~wp:[unit]°C[format]0.0
	{attribute 'OPC.UA.DA' := '1'}
	SP1 AT %M* : REAL := 14; //Gränsvärde start~wp:[unit]°C[format]0.0
END_VAR

	
	IF bInputInvert THEN 
		bProcessedIndication := NOT bIndication;
	ELSE
		bProcessedIndication := bIndication;
	END_IF
	
	IF bSumAlarmConfig THEN
		V := bProcessedIndication AND CMD;
		bAlarm := NOT bProcessedIndication;
	ELSE
		V := bProcessedIndication;
		bAlarm := V XOR CMD;
	END_IF
	
	IF NOT bSafe OR bHandsetBlock THEN
		M := FALSE;
	END_IF;
	
	IF bSumAlarmConfig AND bInputInvert THEN
		PV8 := 'Summalarm NO';
	ELSIF bSumAlarmConfig AND NOT bInputInvert THEN 
		PV8 := 'Summalarm NC'; 
	ELSIF NOT bSumAlarmConfig AND bInputInvert THEN
		PV8 := 'Driftind. inverterad';
	ELSE
		PV8 := 'Driftind.';
	END_IF
	IF bModeHeat THEN
			PV8 := CONCAT('Start Värme, ', PV8);
		ELSE
			PV8 := CONCAT('Start Kyla, ', PV8);
	END_IF

	//Startfördröjning
	fbStartDelay(IN:= (bStart AND bSafe AND NOT bServiceStop), PT:= tStartDelay, Q=> , ET=> );
	bInternalStart := fbStartDelay.Q;

	//Stoppfördröjning
	fbStopDelay(IN:=bIntStart, PT:=INT_TO_TIME(SP3)*60000, Q=>bStart, ET=> );

	//Startar pump om motor är konfigurerad för global pumpmotion 
	IF bPumpmotionConfig THEN
		bPumpMotionStart := oaksGVL.bPumpMotion;
	ELSE
		bPumpMotionStart := FALSE;
	END_IF

	//Digital Utstyrning
	CMD :=  (((bInternalStart OR bPumpMotionStart) AND NOT M) OR (M AND MCMD)) AND bSafe AND NOT bServiceStop;

	//Larm
	fbAlarm1(bInput:=bAlarm , tAlarmDelay:=tAlarmDelay , bAutoReset:=bAutoReset , bAlarmOutput=> AL);
	fbAlarm2(bInput:=M , tAlarmDelay:= , bAutoReset:=TRUE , bAlarmOutput=>AL8 );
	
	//Drifttidsmätning
	fbOperatingHours_1(bEnable:= V, bReset:= RST, rOperatingHours=> PV7 );

	//Justering av SP 	
	IF SP1 < SP2 AND NOT bModeHeat THEN
		SP1 := SP2 + 1;
	ELSIF SP1 > SP2 AND bModeHeat THEN
		SP2 := SP1 + 1;
	END_IF

	//Temp select
	rTempUsed := F_GetTempToUse(rTempToUse);
	
	//Startvillkor temperatur
	IF rTempUsed > SP1 AND NOT bModeHeat THEN
		bIntStart := TRUE;
	ELSIF rTempUsed < SP2 AND NOT bModeHeat THEN
		bIntStart := FALSE;	
	ELSIF (rTempUsed < SP1 OR rTempUsed < 5.0) AND bModeHeat THEN
		bIntStart := TRUE;
	ELSIF (rTempUsed > SP2) AND bModeHeat THEN
		bIntStart := FALSE;	
	END_IF

END_FUNCTION_BLOCK

// oaksLibrary/Utsignal DO_AO/Motorer/fbMotorAo
// "Motorblock" för digital utsignal samt analog utsignal med driftsvar/summalarm med möjlighet att handställa utsignaler. Larmar vid handställning eller utebliven driftindikering/summalarm. 
FUNCTION_BLOCK fbMotorAo EXTENDS fbMotor
VAR_INPUT
	rScaleX1 : REAL := 0; // Ändra om det är 2-10V exempelvis. Max är 0..32767 så 2-10V = 32767 * 0.2 = 6553
	rScaleX2 : REAL := 32767;
	rAnalogInput : REAL; // knyt insignal från exempelvis regulator hit
END_VAR
VAR_OUTPUT
	{attribute 'OPC.UA.DA' := '1'}
	FO_OP AT %Q* : REAL; //Utsignal~wp:[unit]%[format]0[trendoptions]i:300
	{attribute 'OPC.UA.DA' := '1'}
	FO_AL8 AT %M* : BOOL; //Utsignal handställd~wp:[alarmoptions]p:3
END_VAR
VAR
	iTemp4 : INT;
	FB_BA_AO01 : FB_BA_AO;
	
	rY  AT %Q*: REAL;
	TO_iY AT %Q* : INT; 
END_VAR
VAR_INPUT PERSISTENT
	{attribute 'OPC.UA.DA' := '1'}
	FO_M  AT %M*: BOOL; //Handställning~wp:[trendoptions]i:14400, t:1
	{attribute 'OPC.UA.DA' := '1'}
	FO_OPM AT %M*: REAL;//Värde handställning~wp:[unit]%[format]0[trendoptions]i:14400, t:1
END_VAR

SUPER^();

IF NOT bSafe OR bHandsetBlock OR bServiceStop THEN FO_M := FALSE; END_IF

FO_AL8 := FO_M;

IF FO_M THEN
	FO_OP := FO_OPM;
ELSE
	FO_OP := rAnalogInput;	
END_IF

	FB_BA_AO01(
	rX:= FO_OP, 
	rX01:= 0, 
	rX02:= 100, 
	rY01:= rScaleX1, 
	rY02:= rScaleX2 , 
	udiOpMod:= , 
	rXManual:= , 
	rY=> rY, 
	TO_iY=>TO_iY );

// Metod för att sätta analog signal till 0 då CMD ej är till. Knyt denna metod på rAnalogInput:=DIN_MOTOR.mAnalogOutputActiveWhenCmdIsTrue(rDinUtsignal)
METHOD PUBLIC mAnalogOutputActiveWhenCmdIsTrue : REAL
VAR_INPUT
	rSetpoint : REAL;
END_VAR
IF CMD = TRUE THEN
	mAnalogOutputActiveWhenCmdIsTrue := rSetpoint;
ELSE 
	mAnalogOutputActiveWhenCmdIsTrue := 0.0;
END_IF
END_METHOD

END_FUNCTION_BLOCK

// oaksLibrary/Utsignal DO_AO/Motorer/fbMotorAoCool
// Pumpblock för kylshunt. digital utsignal med driftsvar/summalarm med möjlighet att handställa utsignal. Larmar vid handställning eller utebliven driftindikering/summalarm.
// Ibyggd styrning för start/stopp på utetemperatur. OBS!!!!! Använd ej bStart ingång OBS!!!!!
FUNCTION_BLOCK fbMotorAoCool EXTENDS fbMotorAo
VAR_INPUT
	rOutdoorTemp : ANY; //Utetemperatur används för start/stopp Knyter man inget här används oaksGVL.rOutdoortemp
	bCustomStartCon : BOOL := TRUE; //Om ytterligare villkor för start/stopp finns lägg detta här
END_VAR
VAR_OUTPUT
END_VAR
VAR
	fbCoolPumpSr1 : fbCoolPumpSr;
	rTempUsed : REAL; //Uteluftstemperatur
END_VAR
VAR_INPUT PERSISTENT
	{attribute 'OPC.UA.DA' := '1'}
	SP3 AT %M* : INT := 15; //Stoppfördröjning~wp:[unit]min
	{attribute 'OPC.UA.DA' := '1'}
	SP2 AT %M* : REAL := 14;  //Starta pump om utetemp överstiger~wp:[unit]°C[format]0.0
	{attribute 'OPC.UA.DA' := '1'}
	SP1 AT %M* : REAL := 12; //Stoppa pump om utetemp underskrider~wp:[unit]°C[format]0.0
END_VAR

SUPER^();


	//Temp select
	rTempUsed := F_GetTempToUse(rOutdoorTemp);
	
	fbCoolPumpSr1(
	rOutdoorTemp:=rTempUsed , 
	rStartLimit:= SP2, 
	rStopLimit:=SP1 , 
	iStopDelay:=SP3 , 
	bOutput=> );
	
	bStart := fbCoolPumpSr1.bOutput AND bCustomStartCon;

END_FUNCTION_BLOCK

// oaksLibrary/fbCoolPumpSr
// Block för start/stopp på utetemperatur.
// Utgången går till då utetemperatur överstigit inställt värde under inställd tid.
FUNCTION_BLOCK fbCoolPumpSr
VAR_INPUT
	rOutdoorTemp : ANY; // Utetemperatur Knyter man inget här används oaksGVL.rOutdoortemp
END_VAR
VAR_IN_OUT 
	rStartLimit : REAL; // Starta bOutput då rOutdoorTemp underskrider
	rStopLimit : REAL; // Stoppa bOutput då rOutdoorTemp överstiger
	iStopDelay : INT; // Stoppfördröjning
END_VAR
VAR_OUTPUT
	bOutput : BOOL; // Utsignal
	bStopDelayOdt : BOOL; //Stoppfördröjning aktiv via utetemperatur
END_VAR
VAR
	rTempUsed : REAL; // Uteluftstemperatur
	fbPumpTof : TOF;
	bInternalStart : BOOL;
END_VAR

//Temp select
	rTempUsed := F_GetTempToUse(rOutdoorTemp);

IF rStartLimit < rStopLimit THEN
	rStartLimit := rStopLimit + 1;
END_IF

IF rTempUsed > rStartLimit THEN
	bInternalStart := TRUE;
ELSIF rTempUsed < rStopLimit THEN
	bInternalStart := FALSE;	
END_IF

fbPumpTof(IN:=bInternalStart , PT:=INT_TO_TIME(iStopDelay)*60000 , Q=>bOutput , ET=> );

//Stoppfördröjning aktiv
bStopDelayOdt := NOT bInternalStart AND fbPumpTof.Q;

END_FUNCTION_BLOCK

// oaksLibrary/Utsignal DO_AO/Motorer/fbMotorAoRad
// Pumpblock för radiator. digital utsignal med driftsvar/summalarm med möjlighet att handställa utsignal. Larmar vid handställning eller utebliven driftindikering/summalarm.
// Ibyggd styrning för start/stopp på utetemperatur. OBS!!!!! Använd ej bStart ingång OBS!!!!!
FUNCTION_BLOCK fbMotorAoRad EXTENDS fbMotorAo
VAR_INPUT
	rOutdoorTemp : ANY; // Utetemperatur används för start/stopp Knyter man inget här används oaksGVL.rOutdoortemp
	bCustomStartCon : BOOL := TRUE; // Om ytterligare villkor för start/stopp finns lägg detta här
END_VAR
VAR_OUTPUT
END_VAR
VAR
	fbHeatPumpSr1 : fbHeatPumpSr;
	rTempUsed : REAL; //Uteluftstemperatur
END_VAR
VAR_INPUT PERSISTENT
	{attribute 'OPC.UA.DA' := '1'}
	SP3 AT %M* : INT := 15; //Stoppfördröjning~wp:[unit]min
	{attribute 'OPC.UA.DA' := '1'}
	SP2 AT %M* : REAL := 17;  //Stoppa pump om utetemp överstiger~wp:[unit]°C[format]0.0
	{attribute 'OPC.UA.DA' := '1'}
	SP1 AT %M* : REAL := 14; //Starta pump om utetemp underskrider~wp:[unit]°C[format]0.0
END_VAR

SUPER^();

	//Temp select
	rTempUsed := F_GetTempToUse(rOutdoorTemp);

	fbHeatPumpSr1(
	rOutdoorTemp:=rTempUsed , 
	rStartLimit:= SP1, 
	rStopLimit:=SP2 , 
	iStopDelay:=SP3 , 
	bOutput=> );
	
	bStart := fbHeatPumpSr1.bOutput AND bCustomStartCon;

END_FUNCTION_BLOCK

// oaksLibrary/fbHeatPumpSr
// Block för start/stopp på utetemperatur. Utgången går till då utetemp underskrider inställt värde eller fast värde på 5 grader.
// Utgången går från då utetemperatur överstigit inställt värde under inställd tid.
FUNCTION_BLOCK fbHeatPumpSr
VAR_INPUT
	rOutdoorTemp : ANY; // Utetemperatur Knyter man inget här används oaksGVL.rOutdoortemp
END_VAR
VAR_IN_OUT 
	rStartLimit : REAL; // Starta bOutput då rOutdoorTemp underskrider
	rStopLimit : REAL; // Stoppa bOutput då rOutdoorTemp överstiger
	iStopDelay : INT; // Stoppfördröjning
END_VAR
VAR_OUTPUT
	bOutput : BOOL; // Utsignal
	bStopDelayOdt : BOOL; //Stoppfördröjning aktiv via utetemperatur
END_VAR
VAR
	rTempUsed : REAL; // Uteluftstemperatur
	fbPumpTof : TOF;
	bInternalStart : BOOL;
END_VAR

//Temp select
	rTempUsed := F_GetTempToUse(rOutdoorTemp);

IF rStartLimit > rStopLimit THEN
	rStopLimit := rStartLimit + 1;
END_IF

IF rTempUsed < rStartLimit OR rTempUsed < 5.0 THEN
	bInternalStart := TRUE;
ELSIF rTempUsed > rStopLimit THEN
	bInternalStart := FALSE;	
END_IF

fbPumpTof(IN:=bInternalStart , PT:=INT_TO_TIME(iStopDelay)*60000 , Q=>bOutput , ET=> );

//Stoppfördröjning aktiv
bStopDelayOdt := NOT bInternalStart AND fbPumpTof.Q;

END_FUNCTION_BLOCK

// oaksLibrary/Utsignal DO_AO/Motorer/fbMotorAoRl
//"Motorblock" för digital utsignal samt analog utsignal med driftsvar/summalarm med möjlighet att handställa utsignaler. Larmar vid handställning eller utebliven driftindikering/summalarm. 
//Ramptidsbegränsning för analogutgång
FUNCTION_BLOCK fbMotorAoRl EXTENDS fbMotor
VAR_INPUT
	rAnalogInput	: REAL; //knyt insignal från exempelvis regulator hit
	iRampUTime		: INT;	//Max upprampningstid från 0-100% (sek)
	iRampDTime		: INT;	//Max nedrampningstid från 100-0% (sek)
END_VAR
VAR_OUTPUT
	{attribute 'OPC.UA.DA' := '1'}
	FO_OP AT %Q* : REAL; //Utsignal~wp:[unit]%[format]0[trendoptions]i:300
	{attribute 'OPC.UA.DA' := '1'}
	FO_AL8 AT %M* : BOOL; //Utsignal handställd~wp:[alarmoptions]p:3
END_VAR
VAR
	FB_BA_AO01 : FB_BA_AO;
	fbRampLim	: TC3_BA.FB_BA_RampLmt;	
	rFO_OPint	: REAL;
	
	rY  AT %Q*: REAL;
	TO_iY AT %Q* : INT; 
END_VAR
VAR_INPUT PERSISTENT
	{attribute 'OPC.UA.DA' := '1'}
	FO_M  AT %M*: BOOL; //Handställning~wp:[trendoptions]i:14400, t:1
	{attribute 'OPC.UA.DA' := '1'}
	FO_OPM AT %M*: REAL;//Värde handställning~wp:[unit]%[format]0[trendoptions]i:14400, t:1
END_VAR

SUPER^();

FO_AL8 := FO_M;

IF FO_M THEN
	rFO_OPint := FO_OPM;
ELSE
	rFO_OPint := rAnalogInput;	
END_IF

fbRampLim(bEn := TRUE, bEnRamp := TRUE, rIn := rFO_OPint, rHi := 100.0, rLo := 0.0, udiTiUp_sec := INT_TO_UDINT(iRampUTime), udiTiDwn_sec := INT_TO_UDINT(iRampDTime), rOut => FO_OP);

	FB_BA_AO01(
	rX:= FO_OP, 
	rX01:= 0, 
	rX02:= 100, 
	rY01:= 0, 
	rY02:= 32767 , 
	udiOpMod:= , 
	rXManual:= , 
	rY=> rY, 
	TO_iY=>TO_iY );

END_FUNCTION_BLOCK

// oaksLibrary/Utsignal DO_AO/Motorer/fbMotorCool
// Pumpblock för kylshunt. digital utsignal med driftsvar/summalarm med möjlighet att handställa utsignal. Larmar vid handställning eller utebliven driftindikering/summalarm.
// Ibyggd styrning för start/stopp på utetemperatur. OBS!!!!! Använd ej bStart ingång OBS!!!!!
FUNCTION_BLOCK fbMotorCool EXTENDS fbMotor
VAR_INPUT
	rOutdoorTemp : ANY; //Utetemperatur används för start/stopp Knyter man inget här används oaksGVL.rOutdoortemp
	bCustomStartCon : BOOL := TRUE; //Om ytterligare villkor för start/stopp finns lägg detta här
END_VAR
VAR_OUTPUT
END_VAR
VAR
	fbCoolPumpSr1 : fbCoolPumpSr;
	rTempUsed : REAL; //Uteluftstemperatur
END_VAR
VAR_INPUT PERSISTENT
	{attribute 'OPC.UA.DA' := '1'}
	SP3 AT %M* : INT := 15; //Stoppfördröjning~wp:[unit]min
	{attribute 'OPC.UA.DA' := '1'}
	SP2 AT %M* : REAL := 14;  //Starta pump om utetemp överstiger~wp:[unit]°C[format]0.0
	{attribute 'OPC.UA.DA' := '1'}
	SP1 AT %M* : REAL := 12; //Stoppa pump om utetemp underskrider~wp:[unit]°C[format]0.0
END_VAR

SUPER^();

	//Temp select
	rTempUsed := F_GetTempToUse(rOutdoorTemp);
	
	fbCoolPumpSr1(
	rOutdoorTemp:=rTempUsed , 
	rStartLimit:= SP2, 
	rStopLimit:=SP1 , 
	iStopDelay:=SP3 , 
	bOutput=> );
	
	bStart := fbCoolPumpSr1.bOutput AND bCustomStartCon;

END_FUNCTION_BLOCK

// oaksLibrary/Utsignal DO_AO/Motorer/fbMotorHeatBattery
//Oaks AB
//2020-09-28
//Pumpblock för styrning av pump för värmebatteri. Inställbar stoppfördröjning och start då utetemperatur understiger inställt värde. Forcerad start då utetemperatur understiger 5 grader.
//Digital utsignal med driftsvar/summalarm med möjlighet att handställa utsignal. Larmar vid handställning eller utebliven driftindikering/summalarm.
FUNCTION_BLOCK fbMotorHeatBattery EXTENDS fbMotor
VAR_INPUT
	rOutdoorTemp : ANY; //Utetemperatur används för start/stopp Knyter man inget här används oaksGVL.rOutdoortemp
	rValvePos : REAL := 0; //Öppningsgrad värmeventil
END_VAR

VAR_OUTPUT
END_VAR

VAR
	fbHeatPumpSr1 : fbHeatPumpSr;
	rTempUsed : REAL; // Uteluftstemperatur
	bTemp: BOOL;
	rStopLimitInternal : REAL :=6;
END_VAR

VAR_INPUT PERSISTENT
	{attribute 'OPC.UA.DA' := '1'}
	SP1 AT %M* : REAL := 5; //Starta pump om utetemp underskrider~wp:[unit]°C[format]0.0
	{attribute 'OPC.UA.DA' := '1'}
	SP2 AT %M* : REAL := 6;  //Stoppa pump om utetemp överstiger~wp:[unit]°C[format]0.0
	{attribute 'OPC.UA.DA' := '1'}
	SP3 AT %M* : INT := 15; //Stoppfördröjning~wp:[unit]min
END_VAR

	SUPER^();

	//Förhindra för lågt ställd startgräns
	IF SP1 < 5.0 THEN 
		SP1 := 5.0;
	END_IF

	//Start stopp på ventilläge
	IF rValvePos >= 5 THEN
		bTemp := TRUE;
	END_IF;
	
	IF rValvePos = 0 THEN
		bTemp := FALSE;
	END_IF;	
		
	//Temp select
	rTempUsed := F_GetTempToUse(rOutdoorTemp);
	
	//Start stopp på utetemperatur		
	fbHeatPumpSr1(
	rOutdoorTemp:=rTempUsed , 
	rStartLimit:= SP1, 
	rStopLimit:= SP2, 
	iStopDelay:=SP3 , 
	bOutput=> );
	
	bStart := fbHeatPumpSr1.bOutput OR bTemp;
	
	bAutoReset := FALSE; // Ser till så att värmebatteriets pump ej har autoreset.

END_FUNCTION_BLOCK

// oaksLibrary/Utsignal DO_AO/Motorer/fbMotorHiLoSpeed

// "Motorblock" för digital utsignal hel/halvfart med driftsvar/summalarm med möjlighet att handställa utsignal. Larmar vid handställning eller utebliven driftindikering/summalarm.
FUNCTION_BLOCK fbMotorHiLoSpeed
VAR_INPUT
	iStart : INT; //Startvillkor
	bServiceStop : BOOL; //Serviceomkopplare utgång går från om denna ingång är till
	bSafe: BOOL; // Säkerhetsvillkor - Blockerar utsignal i autoläge samt blockerar handställning. Måste vara TRUE för att block ska kunna köras. 
	bAutoReset : BOOL := TRUE; //auto-reset utav driftfel
	bHandsetBlock : BOOL; //Används för blockering av handställning utan att blockera utsignal i autoläge. OBS! - För säkerhetsvillkor se ingång bSafe!
	tAlarmDelay : TIME := T#3S; //Larmfördröjning
	{attribute 'OPC.UA.DA' := '1'}
	RST AT %M* : BOOL := FALSE; //Nollställ drifttid~wp:[trendoptions]i:14400, t:1 
END_VAR
VAR_OUTPUT
	{attribute 'OPC.UA.DA' := '1'}
	CMD AT %M*  : BOOL; //Utsignal~wp:[trendoptions]i:14400, t:1
	{attribute 'OPC.UA.DA' := '1'}
	V AT %M*   : BOOL; //Driftindikering~wp:[trendoptions]i:14400, t:1
	{attribute 'OPC.UA.DA' := '1'}
	AL AT %M* : BOOL; //Driftfel lågfart~wp:
	{attribute 'OPC.UA.DA' := '1'}
	AL1 AT %M* : BOOL; //Driftfel högfart~wp:
	{attribute 'OPC.UA.DA' := '1'}
	AL8 AT %M* : BOOL; //Utsignal handställd~wp:[alarmoptions]p:3
	{attribute 'OPC.UA.DA' := '1'}
	PV1   AT %M* : STRING := ''; //Aktuellt driftläge~wp:
	{attribute 'OPC.UA.DA' := '1'}
	PV4 AT %Q* : BOOL; //Halvfart utsignal~wp:[trendoptions]i:14400, t:1
	{attribute 'OPC.UA.DA' := '1'}
	PV5 AT %Q* : BOOL; //Helfart utsignal~wp:[trendoptions]i:14400, t:1
	bAlarmOutput : BOOL; //internvariabel larm , används för knytning till exempelvis aggregatsblock
	bHandsetOutput : BOOL; //internvariabel handställning, används för knytning till exempelvis aggregatsblock
	{attribute 'OPC.UA.DA' := '1'}
	PV7 AT %M* : UDINT; //Drifttid~wp:[unit]timmar[format]0[trendoptions]i:300 
END_VAR
VAR
	// block för växling från stilla till högfart 
	fbHighSpeedTP : TP;
	fbHighSpeedTon : TON;

	fbLowSpeedTon : TON;
	
	iInternalSpeedMaxValue : INT;
	iInternalSpeedChoice : INT;
	iInternalSpeedValue : INT;
	fbTofBlockLowSpeed : TOF;	
	fbTofBlockHighSpeed : TOF;

	bInternalStartLow : BOOL;
	bInternalStartHigh : BOOL;
	{attribute 'OPC.UA.DA' := '1'}
	V1 AT %I* : BOOL; //Halvfart indikering~wp:[trendoptions]i:14400, t:1
	{attribute 'OPC.UA.DA' := '1'}
	V2 AT %I* : BOOL; //Helfart indikering~wp:[trendoptions]i:14400, t:1
	bProcessedIndication :BOOL; 
	bAlarmLow : BOOL;
	bAlarmHigh : BOOL;
	fbAlarmLow : fbAlarm;
	fbAlarmHigh : fbAlarm;
	fbOperatingHours_1: fbOperatingHours;
END_VAR
VAR_INPUT PERSISTENT
	{attribute 'OPC.UA.DA' := '1'}
	M AT %M* : BOOL; //Handställning~wp:[trendoptions]i:14400, t:1
	{attribute 'OPC.UA.DA' := '1'}
	SP1 AT %M* : INT; //Styrsignal handställning 0 - från 1 - halvfart 2 - helfart~wp:[trendoptions]i:14400, t:1
END_VAR

	IF SP1 < 0 OR SP1 > 2 THEN
		SP1 := 0;
	END_IF

	fbTofBlockLowSpeed(IN:=PV5 , PT:=T#2S , Q=> , ET=> );
	fbTofBlockHighSpeed(IN:=PV4 , PT:=T#2S , Q=> , ET=> );

	AL8 := M;
	
	
	IF NOT bServiceStop AND bSafe THEN
		IF M THEN
			iInternalSpeedMaxValue := SP1; 
		ELSE
			iInternalSpeedMaxValue := iStart; 
		END_IF
	ELSE
		iInternalSpeedMaxValue := 0; 	
	END_IF;
	
	// Växling från stillastående till halvfart
	IF iInternalSpeedMaxValue = 1 AND iInternalSpeedChoice = 0 THEN 
		iInternalSpeedValue := 1;
		iInternalSpeedChoice := 1;
	END_IF;
	
	// Växling från stillastående till helfart
	fbHighSpeedTP(PT:=T#10S);
	fbHighSpeedTon(PT:=T#2S);
	IF iInternalSpeedMaxValue = 2 AND iInternalSpeedChoice = 0 THEN 
		fbHighSpeedTP(IN := TRUE);
		fbHighSpeedTon(IN := FALSE);
		iInternalSpeedValue := 1;
		iInternalSpeedChoice := 1;
	ELSIF iInternalSpeedMaxValue = 2 AND NOT fbHighSpeedTP.Q THEN
		fbHighSpeedTon.IN := TRUE;
		IF fbHighSpeedTon.Q THEN
			iInternalSpeedValue := 2;
			iInternalSpeedChoice := 2;
		ELSE
			iInternalSpeedValue := 0;
			iInternalSpeedChoice := -1;
		END_IF;
		fbHighSpeedTP.IN := FALSE;
	END_IF;
	// Växling från högfart till lågfart
	fbLowSpeedTon(PT:=T#2S);
	IF iInternalSpeedMaxValue = 1 AND iInternalSpeedChoice = 2 THEN 
		iInternalSpeedValue := 0;
		fbLowSpeedTon(IN := TRUE);
		IF fbLowSpeedTon.Q THEN
			iInternalSpeedValue := 1;
			iInternalSpeedChoice := 1;
		END_IF
	ELSE
		fbLowSpeedTon(IN := FALSE);
	END_IF;
	
	// Växling till stillastående
	IF  iInternalSpeedMaxValue = 0 THEN 
		iInternalSpeedValue := iInternalSpeedMaxValue;
		iInternalSpeedChoice := 0;
	END_IF;
	

	
	
	bProcessedIndication := V1 OR V2;
	V := bProcessedIndication;
	
	IF NOT bSafe OR bHandsetBlock THEN
		M := FALSE;
	END_IF;
	
	
	
	//bHandsetLowSpeed :=  ;
	//bHandsetHighSpeed := ;
(*	
	IF NOT  bInternalStartLow AND NOT bInternalStartHigh AND (iStart = 2 OR SP1 = 2) THEN
		iInternalSpeedValue := 1;
		
	
	END_IF
*)
	
	bInternalStartLow := iInternalSpeedValue =1;
	bInternalStartHigh := iInternalSpeedValue =2;
	

	
	IF PV4 THEN
		PV1 := 'Halvfart';
	ELSIF PV5 THEN
		PV1 := 'Helfart';
	ELSE
		PV1 := 'Utsignal från';
	END_IF
	
	PV4 :=  ((bInternalStartLow) AND NOT bServiceStop) AND bSafe AND NOT fbTofBlockLowSpeed.Q;
	
	PV5 :=  ((bInternalStartHigh) AND NOT bServiceStop) AND bSafe AND NOT fbTofBlockHighSpeed.Q;
	
	CMD := PV4 OR PV5;
	V := V1 OR V2;


	bAlarmLow := PV4 XOR V1;
	bAlarmHigh := PV5 XOR V2;
	
	fbAlarmLow(bInput:=bAlarmLow , tAlarmDelay:=tAlarmDelay , bAutoReset:=bAutoReset , bAlarmOutput=> AL);
	fbAlarmHigh(bInput:=bAlarmHigh , tAlarmDelay:=tAlarmDelay , bAutoReset:=bAutoReset , bAlarmOutput=> AL1);
	
	bAlarmOutput := AL OR AL1;
	bHandsetOutput := INT_TO_BOOL(SP1);

	//Drifttidsmätning
	fbOperatingHours_1(bEnable:= V, bReset:= RST, rOperatingHours=> PV7 );

END_FUNCTION_BLOCK

// oaksLibrary/Utsignal DO_AO/Motorer/fbMotorRad
// Pumpblock för radiator. digital utsignal med driftsvar/summalarm med möjlighet att handställa utsignal. Larmar vid handställning eller utebliven driftindikering/summalarm.
// Ibyggd styrning för start/stopp på utetemperatur. OBS!!!!! Använd ej bStart ingång OBS!!!!!
FUNCTION_BLOCK fbMotorRad EXTENDS fbMotor
VAR_INPUT
	rOutdoorTemp : ANY; // Utetemperatur används för start/stopp Knyter man inget här används oaksGVL.rOutdoortemp
	bCustomStartCon : BOOL := TRUE; // Om ytterligare villkor för start/stopp finns lägg detta här
END_VAR
VAR_OUTPUT
END_VAR
VAR
	fbHeatPumpSr1 : fbHeatPumpSr;
	rTempUsed : REAL; // Uteluftstemperatur
END_VAR
VAR_INPUT PERSISTENT
	{attribute 'OPC.UA.DA' := '1'}
	SP3 AT %M* : INT := 15; //Stoppfördröjning~wp:[unit]min
	{attribute 'OPC.UA.DA' := '1'}
	SP2 AT %M* : REAL := 17;  //Stoppa pump om utetemp överstiger~wp:[unit]°C[format]0.0
	{attribute 'OPC.UA.DA' := '1'}
	SP1 AT %M* : REAL := 14; //Starta pump om utetemp underskrider~wp:[unit]°C[format]0.0
END_VAR

SUPER^();

	//Temp select
	rTempUsed := F_GetTempToUse(rOutdoorTemp);
	
	fbHeatPumpSr1(
	rOutdoorTemp:=rTempUsed , 
	rStartLimit:= SP1, 
	rStopLimit:=SP2 , 
	iStopDelay:=SP3 , 
	bOutput=> );
	
	bStart := fbHeatPumpSr1.bOutput AND bCustomStartCon;

END_FUNCTION_BLOCK

// oaksLibrary/Utsignal DO_AO/Motorer/fbTwinMotorControl
// parpumpsblock ej klart
FUNCTION_BLOCK fbTwinMotorControl
VAR_INPUT
	{attribute 'OPC.UA.DA' := '1'}
	V AT %M* : BOOL; //Startsignal~wp:[trendoptions]i:14400, t:1
	bError1,bError2 : BOOL;
	{attribute 'OPC.UA.DA' := '1'}
	M AT %M*  : BOOL; //Manuell pumpväxling~wp:[trendoptions]i:14400, t:1
END_VAR
VAR_OUTPUT
	{attribute 'OPC.UA.DA' := '1'}
	PV AT %M* : INT; //Aktuellt pumpval~wp:[trendoption]i:300
	bStartOutput1,bStartOutput2 : BOOL;
	{attribute 'OPC.UA.DA' := '1'}
	AL AT %M* : BOOL; //Driftfel parpumpar~wp:
END_VAR
VAR 
	wLastDayOfChange: WORD;
	fbDayTrig: R_trig;
	
	itemp : int;
	
	stTime		: tc2_ba.TIMESTRUCT;
	nActualDayCase	: INT;
	nActualHour 	: INT;
	nActualMinute 	: INT;
	
	FB_BA_GetTime01 : tc2_ba.FB_BA_GetTime; 
	FB_BA_ExtTiSt01 : tc2_ba.FB_BA_ExtTiSt;	
	
	
	nTime : INT; // Internvariabel aktuell tid (nActualHour+nActualMinute)
	
	bDay : BOOL; // Internvariabel blir TRUE om inställd dag är lika med aktuell dag
	bTime : BOOL; // Internvariabel blir TRUE om inställd tid är lika med aktuell tid
	
	fbHandsetToN: TON;
	fbAlarm1 : fbAlarm;
END_VAR
VAR_INPUT PERSISTENT
	{attribute 'OPC.UA.DA' := '1'}
	SP1 AT %M*  : INT:=1; //Dag för pumpväxling (-1 = ingen växling 0 = Söndag 1 = Måndag 2 = Tisdag..6 = Söndag~wp:
	{attribute 'OPC.UA.DA' := '1'}
	SP2 AT %M*  : INT:=1000; //Tid för pumpväxling~wp:[format]00:00[engmin]0[engmax]2400
END_VAR

	fbHandsetToN.PT := T#1S;
	fbHandsetToN(IN:=M);
	
	IF fbHandsetToN.Q THEN 
		M := FALSE;
	END_IF

	FB_BA_GetTime01(bEn :=TRUE);	
	stTime := FB_BA_GetTime01.stSysTi;

	nActualDayCase :=WORD_TO_INT (stTime.wDayOfWeek);
	nActualHour :=WORD_TO_INT (stTime.wHour)*100;
	nActualMinute :=WORD_TO_INT (stTime.wMinute);
	
	// nActualHour+nActualMinute
	
	nTime := nActualHour+nActualMinute;
	
	bDay := nActualDayCase = SP1;
	bTime := nTime = SP2;


	IF SP1 < -1 OR  SP1>7 THEN
		SP1 := 1;
	END_IF
	
	IF SP2 < 0 OR  SP2>2359 THEN
		SP2 := 1200;
	END_IF

	IF PV < 1 OR PV > 2  THEN	
		PV := 1;
	END_IF;

	
	IF (bDay AND bTime) OR M THEN
		fbDayTrig(CLK := TRUE);
	ELSE
		fbDayTrig(CLK := FALSE);
	END_IF

	IF fbDayTrig.Q THEN
		IF PV = 1 THEN
			PV := 2;
		ELSE
			PV := 1;
		END_IF
	END_IF
	
	bStartOutput1 := ((PV = 1 AND NOT bError1) OR bError2) AND V;
	bStartOutput2 := ((PV = 2 AND NOT bError2) OR bError1) AND V;

	fbAlarm1(bInput:= bError1 AND bError2 , tAlarmDelay:= T#3S , bAutoReset:=TRUE , bAlarmOutput=> AL);

END_FUNCTION_BLOCK

// oaksLibrary/Utsignal DO_AO/Motorer/fbTwinMotorControlCool
// Pumpblock för radiator. digital utsignal med driftsvar/summalarm med möjlighet att handställa utsignal. Larmar vid handställning eller utebliven driftindikering/summalarm.
// Ibyggd styrning för start/stopp på utetemperatur. OBS!!!!! Använd ej bStart ingång OBS!!!!!
FUNCTION_BLOCK fbTwinMotorControlCool EXTENDS fbTwinMotorControl
VAR_INPUT
	rOutdoorTemp : ANY; //Utetemperatur används för start/stopp Knyter man inget här används oaksGVL.rOutdoortemp
	bCustomStartCon : BOOL := TRUE; //Om ytterligare villkor för start/stopp finns lägg detta här
END_VAR
VAR_OUTPUT
END_VAR
VAR
	rTempUsed : REAL; //Uteluftstemperatur
	fbCoolPumpSr1 : fbCoolPumpSr;
END_VAR
VAR_INPUT PERSISTENT
	{attribute 'OPC.UA.DA' := '1'}
	SP5 AT %M* : INT := 15; //Stoppfördröjning~wp:[unit]min
	{attribute 'OPC.UA.DA' := '1'}
	SP4 AT %M* : REAL := 14;  //Starta pump om utetemp överstiger~wp:[unit]°C[format]0.0
	{attribute 'OPC.UA.DA' := '1'}
	SP3 AT %M* : REAL := 12; //Stoppa pump om utetemp underskrider~wp:[unit]°C[format]0.0
END_VAR

SUPER^();
	//Temp select
	rTempUsed := F_GetTempToUse(rOutdoorTemp);

	fbCoolPumpSr1(
	rOutdoorTemp:=rTempUsed , 
	rStartLimit:= SP4, 
	rStopLimit:= SP3  , 
	iStopDelay:=SP5 , 
	bOutput=> );
	
	V := fbCoolPumpSr1.bOutput AND bCustomStartCon;

END_FUNCTION_BLOCK

// oaksLibrary/Utsignal DO_AO/Motorer/fbTwinMotorControlRad
// Pumpblock för radiator. digital utsignal med driftsvar/summalarm med möjlighet att handställa utsignal. Larmar vid handställning eller utebliven driftindikering/summalarm.
// Ibyggd styrning för start/stopp på utetemperatur. OBS!!!!! Använd ej bStart ingång OBS!!!!!
FUNCTION_BLOCK fbTwinMotorControlRad EXTENDS fbTwinMotorControl
VAR_INPUT
	rOutdoorTemp : ANY; //Utetemperatur används för start/stopp Knyter man inget här används oaksGVL.rOutdoortemp
	bCustomStartCon : BOOL := TRUE; //Om ytterligare villkor för start/stopp finns lägg detta här
END_VAR
VAR_OUTPUT
END_VAR
VAR
	fbHeatPumpSr1 : fbHeatPumpSr;
	rTempUsed : REAL; //Uteluftstemperatur
END_VAR
VAR_INPUT PERSISTENT
	{attribute 'OPC.UA.DA' := '1'}
	SP5 AT %M* : INT := 15; //Stoppfördröjning~wp:[unit]min
	{attribute 'OPC.UA.DA' := '1'}
	SP4 AT %M* : REAL := 17;  //Stoppa pump om utetemp överstiger~wp:[unit]°C[format]0.0
	{attribute 'OPC.UA.DA' := '1'}
	SP3 AT %M* : REAL := 14; //Starta pump om utetemp underskrider~wp:[unit]°C[format]0.0
END_VAR

SUPER^();

	//Temp select
	rTempUsed := F_GetTempToUse(rOutdoorTemp);
	
	fbHeatPumpSr1(
	rOutdoorTemp:=rTempUsed , 
	rStartLimit:= SP3, 
	rStopLimit:=SP4 , 
	iStopDelay:=SP5 , 
	bOutput=> );
	
	V := fbHeatPumpSr1.bOutput AND bCustomStartCon;

END_FUNCTION_BLOCK

// oaksLibrary/Utsignal DO_AO/Värmeväxling/Enskilda funktioner/fbCoolRecycleHeatExhanger
//Funktionsblock för kylåtervinning. 
//Funktion är aktiv då fläktindikering är till samt frånluftstemperatur understiger uteluftstemperatur med 1°C. Funktion avvaktiveras utetemperatur är lägre är frånluftstemperatur.
FUNCTION_BLOCK fbCoolRecycleHeatExhanger
VAR_INPUT
bSupFanInd : BOOL; //Driftindikering tilluftsfläkt
rOutdoorTemp : ANY; //Uteluftstemperatur Knyter man inget här används oaksGVL.rOutdoortemp
rExhTemp : REAL; //Frånluftstemperatur
END_VAR
VAR_OUTPUT
	{attribute 'OPC.UA.DA' := '1'}
	V AT %M* : BOOL; //Kylåtervinning~wp:[trendoptions]i:14400, t:1
END_VAR
VAR
	rTempUsed : REAL; //Uteluftstemperatur
END_VAR


//Temp select
rTempUsed := F_GetTempToUse(rOutdoorTemp);
	

IF bSupFanInd AND rTempUsed > (rExhTemp + 1) THEN
	V := TRUE;
END_IF
IF bSupFanInd = FALSE OR rTempUsed < rExhTemp THEN
	V := FALSE;
END_IF

END_FUNCTION_BLOCK

// oaksLibrary/Utsignal DO_AO/Värmeväxling/Enskilda funktioner/fbHeatExchangerStartup
// uppstartsblock vvx för ventilationsaggregat. Startar VVX på 100% OM frånluftsfläkt är till, tilluftsfläkt är från och utetemp är under 5 grader. Utetempsvillkoret är frånslagsfördröjt med 2 minuter.
FUNCTION_BLOCK fbHeatExchangerStartup
VAR_INPUT
	bSupfanIndication : BOOL; // driftindikering tilluftsfläkt
	bExhfanIndication : BOOL; // driftindikering frånluftsfläkt
	rOutdoortemp : ANY; // utetemp Knyter man inget här används oaksGVL.rOutdoortemp
	rControllerSignal : REAL; // regulatorsignal knyts hit
END_VAR
VAR_OUTPUT
	rOutput : REAL; // utgång knyts till vvx ingång
END_VAR
VAR
	fbOutdoortempTof : TOF;
	rTempUsed : REAL; // Uteluftstemperatur
END_VAR


//Temp select
rTempUsed := F_GetTempToUse(rOutdoorTemp);

fbOutdoortempTof(IN:=rTempUsed < 5.0 AND bExhfanIndication , PT:= T#2M , Q=> , ET=> );

IF bSupfanIndication THEN
	rOutput := rControllerSignal;
ELSIF bExhfanIndication AND fbOutdoortempTof.Q THEN
	rOutput :=  100;
ELSE
	rOutput := 0;
END_IF

END_FUNCTION_BLOCK

// oaksLibrary/Utsignal DO_AO/Värmeväxling/Korsvärmeväxlare/fbCrossFlowHeatExchanger
// Block för kors-vvx. avfrostningsfunktion med digital tryckvakt
FUNCTION_BLOCK fbCrossFlowHeatExchanger EXTENDS fbAnalogSignalLogic
VAR_INPUT
	bInvertGpIndication : BOOL; // invertera signal för digital tryckvakt
END_VAR
VAR_OUTPUT
	{attribute 'OPC.UA.DA' := '1'}
	GP_AL AT %M* : BOOL; //Lång avfrostning VVX~wp:
	{attribute 'OPC.UA.DA' := '1'}
	GP_V AT %M* : BOOL; //Indikering tryckvakt~wp:
	{attribute 'OPC.UA.DA' := '1'}
	GP_PV AT %M* : STRING; //Statustext avfrostning~wp:
	{attribute 'OPC.UA.DA' := '1'}
	DEFROST_V AT %M* : BOOL; //Indikering avfrostning~wp:[trendoptions]i:14400, t:1
	{attribute 'OPC.UA.DA' := '1'}
	INV_OP AT %M* : REAL;//Fiktiv inverterad signal för visning i webport~wp:[unit]%[format]0[trendoptions]i:300
END_VAR
VAR
	fbDefrostAlarm : fbAlarm;
	bGpIndication AT %I* : BOOL; // digital tryckvakt för io-knytning
	fbDefrostTof : TOF; // frånslagsfördröjning avfrostning VVX
END_VAR

VAR_INPUT PERSISTENT
	{attribute 'OPC.UA.DA' := '1'}
	GP_SP1 AT %M* : REAL := 50; //Utsignal återvinning vid avfrostning~wp:[unit]%[format]0
	{attribute 'OPC.UA.DA' := '1'}
	GP_SP2 AT %M* : INT := 5; //Minsta tid avfrostning~wp:[unit]minuter[format]0
	{attribute 'OPC.UA.DA' := '1'}
	GP_AD AT %M* : INT :=60;//Larmfördröjning lång avfrostning~wp:[unit]minuter[format]0
END_VAR

SUPER^();

IF bInvertGpIndication THEN
	GP_V := NOT bGpIndication;
ELSE
	GP_V := bGpIndication;
END_IF

// Avfrostningsindikering frånslagsfördröjd (används för att styra ner återvinning VVX)
fbDefrostTof(IN:=GP_V , PT:=INT_TO_TIME(GP_SP2)*60000 , Q=>DEFROST_V , ET=> );

fbDefrostAlarm(bInput:=DEFROST_V , tAlarmDelay:=INT_TO_TIME(GP_AD)*60000 , bAutoReset:=TRUE , bAlarmOutput=>GP_AL );

// Vid avfrostning styr om VVX-signal till inställingsvärde
IF DEFROST_V AND NOT M THEN
	OP := GP_SP1;
END_IF

IF DEFROST_V THEN
	GP_PV := 'Avfrostning VVX aktiv';
ELSE
	GP_PV := ' ';
END_IF

INV_OP := 100 - OP;

END_FUNCTION_BLOCK

// oaksLibrary/Utsignal DO_AO/Värmeväxling/Korsvärmeväxlare/fbCrossFlowHeatExhTemp
//Funktionsblock för avfrostning av korsvärmeväxlare/plattvärmeväxlare med by-pass spjäll. Då utetemperatur och verkningsgrad understiger inställt värde och starfördröjning har löpt ut sker avfrostning under inställd tid.
//SP6 skapas utanför block för att ange tex Pa/%/l/s. 
FUNCTION_BLOCK fbCrossFlowHeatExhTemp EXTENDS fbAnalogSignalLogic
VAR_INPUT
bExhfan : BOOL; //Driftindikering frånluftsfläkt 
rOutdoorTemp : ANY; //Ute-/kanaltemperatur Knyter man inget här används oaksGVL.rOutdoortemp
rHeatEfficency : REAL; //Verkninsgrad
END_VAR
VAR_OUTPUT
	{attribute 'OPC.UA.DA' := '1'}
	V AT %M* : BOOL; //Avfrostning aktiv~wp:[trendoptions]i:300[trendoptions]i:14400, t:1
	{attribute 'OPC.UA.DA' := '1'}
	AL AT %M* : BOOL; //Lång avfrostningstid~wp:
	{attribute 'OPC.UA.DA' := '1'}
	INV_OP AT %M* : REAL;//Fiktiv inverterad signal för visning i webport~wp:[unit]%[format]0[trendoptions]i:300
END_VAR
VAR
	rTempUsed : REAL; // Uteluftstemperatur
	bStart : BOOL; //Startvillkor
	bRestart : BOOL; //Omstart
	fbStartDelay: TON;
	fbDefrost: TP;
	fbAlarm: fbalarm;
END_VAR
VAR_INPUT PERSISTENT
	{attribute 'OPC.UA.DA' := '1'}
	SP1 AT %M* : INT :=0;//Startgräns då utetemperatur understiger~wp:[unit]°C[format]0.0
	{attribute 'OPC.UA.DA' := '1'}
	SP2 AT %M* : INT :=30;//Starta avfrostning då verkningsgrad understiger~wp:[unit]%[format]0
	{attribute 'OPC.UA.DA' := '1'}
	SP3 AT %M* : INT :=5;//Startfördröjning avfrostning~wp:[unit]minuter[format]0
	{attribute 'OPC.UA.DA' := '1'}
	SP4 AT %M* : INT :=10;//Frånslagsfördröjning avfrostning~wp:[unit]minuter[format]0
	{attribute 'OPC.UA.DA' := '1'}
	SP5 AT %M* : INT :=60;//Fördröjning lång avfrostning~wp:[unit]minuter[format]0
END_VAR

	SUPER^();
	
	
//Temp select
rTempUsed := F_GetTempToUse(rOutdoorTemp);
//Villkor
bStart := (rTempUsed < SP1) AND (rHeatEfficency < SP2) AND bExhfan; 

//Reset avfrostning vid avstängd fläkt
IF bExhfan THEN
	fbDefrost.PT := INT_TO_TIME(SP4)*60000;
ELSE
	fbDefrost.PT := T#0S;
END_IF

//Startfördröjning
IF bStart AND bRestart THEN 
	fbStartDelay.IN := TRUE;
ELSE
	fbStartDelay.IN := FALSE;
END_IF

fbStartDelay(IN:= , PT:= INT_TO_TIME(SP3)*60000, Q=> , ET=> );

//Avfrostning
fbDefrost(IN:=fbStartDelay.Q, 
PT:=, //Tid ställs från startvillkor
Q=>,
ET=> 
);

IF fbDefrost.Q THEN
	V := TRUE;
	bRestart := FALSE; 
ELSE
	V := FALSE;
	bRestart := TRUE;
END_IF

//Larm lång avfrostning
fbAlarm(bInput:= bStart, tAlarmDelay:=INT_TO_TIME(SP5)*60000, bAutoReset:= TRUE, bAlarmOutput=> AL);

// Vid avfrostning styr om VVX-signal till inställingsvärde
IF V AND NOT M THEN
	OP := 0;
END_IF

INV_OP := 100 - OP;

END_FUNCTION_BLOCK

// oaksLibrary/Utsignal DO_AO/Värmeväxling/fbHeatExhange
///Oaks AB
//2020-10-06
//Funktionsblock för styrning återvinning med inbyggd kylåtervinning och förberedd uppstart.
//Kan användas till både, roterande värmeväxlare, korsvärmeväxlare med by-pass och vätskeburen återvinning (min.begränsning).

FUNCTION_BLOCK fbHeatExhange
VAR_INPUT
	//Generella
	rProcessValue : REAL; //Insignal från regulator
	bSupfanIndication : BOOL; //Driftindikering tilluftsfläkt
	bExhfanIndication : BOOL; //Driftindikering frånluftsfläkt
	//Minbegränsning returtemperatur
	bEnableReturnTempLim : BOOL :=FALSE;//Använd returbegränsning vätskeburen återvinning
	rReturnTemp : REAL :=0; //Returtemperatur vätskeburen återvinning
	rReturnTempLim : REAL :=0; //Min.begränsning returtemperatur vätskeburen återvinning
	
	rReturnTempLimKp : REAL :=20; //Kp returbegränsning
	rReturnTempLimKi : UDINT :=5; //Ki returbegränsning
	
	//Temperaturer
	rOutdoorTemp : REFERENCE TO REAL; //Uteluftstemperatur Knyter man inget här används oaksGVL.rOutdoortemp
	rExhTemp : REAL :=0; //Frånluftstemperatur
	bEnableCoolRecycle : BOOL :=FALSE; //Använd kylåtervinning
	rOutdoorTempStartup : REAL := 10; //Gräns utetemperatur förberedd uppstart
END_VAR
VAR_OUTPUT
	rOutput : REAL; //Utsignal
	bCoolRecycle : BOOL ; //Aktiv kylåtervinning
	bPumpStart AT %M* : BOOL; //Pumpstart vid vätskeburen återvinning (OP >= 5)
END_VAR
VAR
	rTempUsed : REAL; // Uteluftstemperatur
	fbReg01 : Tc3_BA_Common.FB_BA_PIDCtrl;
	fbOutdoortempTof : TOF;

	rOutputStartDelay : REAL; //Utsignal från förberedd uppstart
	rOutputCoolRecycle : REAL; //Utsignal från kylåtervinning
	rReturnTempOutput : REAL; //Utsignal från min.begräsning returtemperatur
END_VAR

//Generellt
	//Temp select
	IF __ISVALIDREF(rOutdoorTemp) THEN
		rTempUsed := rOutdoorTemp;
	ELSE
		rTempUsed := oaksGVL.rOutdoorTemp;
	END_IF
		
	//Uppstart
	fbOutdoortempTof(IN:=rTempUsed < rOutdoorTempStartup AND bExhfanIndication , PT:= T#2M , Q=> , ET=> );
	
	IF bSupfanIndication THEN
		rOutputStartDelay := rProcessValue;
	ELSIF bExhfanIndication AND fbOutdoortempTof.Q THEN
		rOutputStartDelay :=  100;
	ELSE
		rOutputStartDelay := 0;
	END_IF

	//Kylåtervinning
	IF bSupfanIndication AND rTempUsed > (rExhTemp + 1) AND rProcessValue = 0 AND bEnableCoolRecycle THEN
		bCoolRecycle := TRUE;
		rOutputCoolRecycle := 100;
	END_IF
	IF bSupfanIndication = FALSE OR rTempUsed < rExhTemp OR rProcessValue > 1 OR NOT bEnableCoolRecycle THEN
		bCoolRecycle := FALSE;
		rOutputCoolRecycle := 0;
	END_IF
	
//Vätskeåtervinning
	fbReg01(
	bEn:=bExhfanIndication AND bEnableReturnTempLim, 
	rW:=rReturnTempLim , 
	rX:=rReturnTemp, 
	udiOpMode:= , 
	bActn:= TRUE, 
	rKp:= rReturnTempLimKp, 
	udiTn_ms:= rReturnTempLimKi * 1000, 
	udiTv_ms:= , 
	udiTd_ms:= , 
	rYMax:=100 , 
	rYMin:= 0, 
	rNZ:= , 
	udiCycCl:= , 
	bSync:= , 
	rSync:= , 
	rY=> , 
	rE=> , 
	bARW=> );
	
	IF bEnableReturnTempLim AND bExhfanIndication THEN
		rReturnTempOutput := fbReg01.rY;
	ELSE
		rReturnTempOutput := 100;
	END_IF

	//Pumpstart
	IF MAX(rOutputStartDelay,rProcessValue,rOutputCoolRecycle) >= 5 AND bEnableReturnTempLim THEN
		bPumpStart := TRUE;
	END_IF
	
	IF MAX(rOutputStartDelay,rProcessValue,rOutputCoolRecycle) = 0 OR NOT bEnableReturnTempLim THEN
		bPumpStart := FALSE;
	END_IF

	
//Utsignal 
 rOutput := MIN(MAX(rOutputStartDelay,rProcessValue,rOutputCoolRecycle), rReturnTempOutput);

END_FUNCTION_BLOCK

// oaksLibrary/Utsignal DO_AO/Värmeväxling/fbHeatExhangeEff
///Oaks AB
//2020-10-06
//Funktionsblock för styrning återvinning med inbyggd verkningsgrad kylåtervinning och förberedd uppstart.
//Kan användas till både, roterande värmeväxlare, korsvärmeväxlare med by-pass och vätskeburen återvinning (min.begränsning).
//Verkningsgrad = (Tilluft efter VVX - Uteluft) / (Frånluft - Uteluft)
//Verkningsgrad = (Frånluft efter VVX - Avluft) / (Frånluft - Uteluft)
FUNCTION_BLOCK fbHeatExhangeEff EXTENDS fbHeatExhange
VAR_INPUT
	//Temperaturer
	rSupTemp : REAL; //Tilluftstemperatur efter VVX
	rExhaustTemp : REAL; //Avluftstemperatur
	//Verkningsgrad
	bEfficencyType : BOOL; //TRUE = Tilluft efter VVX/frånluft/uteluft FALSE= Frånluft/avluft/uteluft
END_VAR

VAR_INPUT PERSISTENT
	{attribute 'OPC.UA.DA' := '1'}
	AD AT %M* : INT :=60; //Larmfördröjning~wp:[unit]minuter[format]0
	{attribute 'OPC.UA.DA' := '1'}
	ALL AT %M* : INT :=30; //Låg gräns verkningsgrad~wp:[unit]%[format]0
	{attribute 'OPC.UA.DA' := '1'}
	AHL AT %M* : INT :=90; //Hög gräns verkningsgrad~wp:[unit]%[format]0
END_VAR

VAR_OUTPUT
	//Verkningsgrad
	{attribute 'OPC.UA.DA' := '1'}
	PV AT %M* : REAL; //Verkningsgrad~wp:[unit]%[format]0[trendoption]i:300
	{attribute 'OPC.UA.DA' := '1'}
	LAL AT %M* : BOOL; //Låg verkningsgrad~wp:
	{attribute 'OPC.UA.DA' := '1'}
	HAL AT %M* : BOOL; //Hög verkningsgrad~wp:
END_VAR

VAR
	itemp : int;
	rEff : REAL;
	rTemp : REAL; // Tempvariablel
	fbLowEffeciency : fbLowLimitAlarm;
	fbHighEffeciency : fbHighLimitAlarm;
	bCalcAtive : BOOL;
END_VAR

	SUPER^();	
	//Verkningsgrad
	rTemp := rExhTemp-rTempUsed;
		
	//Aktivering av beräkning
	IF rOutput > 0 THEN
		bCalcAtive := TRUE;
	ELSE
		bCalcAtive := FALSE;
	END_IF;
		
	IF bEfficencyType AND rTemp <> 0 AND NOT bCoolRecycle AND bSupfanIndication AND bCalcAtive THEN
		rEff := ((rSupTemp-rTempUsed)/rTemp)*100;
	ELSIF bEfficencyType = FALSE AND rTemp <> 0 AND NOT bCoolRecycle AND bSupfanIndication AND bCalcAtive THEN
		rEff := ((rExhTemp-rExhaustTemp)/rTemp)*100;
	ELSIF bCoolRecycle OR NOT bSupfanIndication OR NOT bCalcAtive THEN
		rEff := 0;
	END_IF
	
	IF rEff > 100 THEN
		PV := 100;
	ELSIF rEff < 0 THEN
		PV := 0;
	ELSE
		PV := rEff;
	END_IF
	
		// Larmfunktion låg/hög verkningsgrad
		fbLowEffeciency(
			//bInput:= , 
			tAlarmDelay:= INT_TO_TIME(AD)*60000, 
			bAutoReset:=TRUE, 
			bAlarmOutput=>LAL, 
			bEnable:= rProcessValue = 100 AND NOT bCoolRecycle, 
			rProcessValue:=PV, 
			rLowLimit:=ALL
		);
		fbHighEffeciency(
			//bInput:= , 
			tAlarmDelay:= INT_TO_TIME(AD)*60000, 
			bAutoReset:= TRUE, 
			bAlarmOutput=>HAL , 
			bEnable:= rProcessValue = 100 AND NOT bCoolRecycle, 
			rProcessValue:=PV, 
			rHighLimit:=AHL 
		);

END_FUNCTION_BLOCK

// oaksLibrary/Utsignal DO_AO/fbAnalogSignalLogicFb
//Block för analoga utsignaler med möjlighet att handställa utsignal. Larmar vid handställning.
//Ingång för lägesåterföring (feedback) för visning samt generering av larm om avvikelse mellan OP och MV (feedback) är större än gräns
FUNCTION_BLOCK fbAnalogSignalLogicFb
VAR_INPUT
	//Analogutgång
	rSetpoint 	: REAL; 			//Insginal för auto-läge (exmepelvis regulatorsignal)
	bInterlock 	: BOOL; 			//blockering av handställning
	bInvert 	: BOOL := FALSE; 	//Invertering utgång
	
	//Analogingång (feedback)
	AIrScaleX1 	: REAL; 				//Ändra om det är 2-10V exempelvis. Max är 0..32767 så 2-10V = 32767 * 0.2 = 6553
	AIrScaleX2 	: REAL := 32767;
	AIrScaleMin : REAL;
	AIrScaleMax : REAL;
	AIiBusTermType : E_BA_TERMINAL_KL := 17; //Bus-terminal typ AI
	AI_M AT %M* : BOOL;					//Handställning återföring~wp:
END_VAR
VAR_OUTPUT
	//Analogutgång
	OP AT %M* 		: REAL;  	//Utsignal~wp:[unit]%[format]0.0[trendoptions]i:60
	AL8 AT %M* 		: BOOL;		//Utsignal handställd~wp:[alarmoptions]p:3
	
	//Analogingång
	PV AT %M*  		: REAL;		//Återföring~wp:[unit]%[format]0.0[trendoptions]i:60
	FAULT AT %M* 	: BOOL;		//Signalfel återföring~wp:
	
	AL AT %M* 		: BOOL;		//Konfliktlarm~wp:[alarmoptions]p:3
END_VAR
VAR
	rOPold			: REAL;		//Hjälpvariabel för att avvakta stadig reglersignal	

	//Analogutgång
	FB_BA_AO01 		: FB_BA_AO;
	rY  AT %Q*		: REAL;
	TO_iY AT %Q* 	: INT; 
	rOutputInternal : REAL;	 	//Intern signal för invertering/ej invertering
	
	fbAlarm2 	: fbAlarm; 		//Larm handställning
	fbAlarmFb 	: fbAlarm; 		//Larm återföring
	
	//Analogingång
	usiState AT %I*		: USINT;
	iDataIn AT %I*		: INT;
	usiCtrl AT %Q*		: USINT;
	iDataOut AT %Q*		: INT;
	FB_BA_AI01 			: FB_BA_AI;
	FB_BA_TiAvrg01 		: tc2_ba.FB_BA_TiAvrg;
END_VAR
VAR_INPUT PERSISTENT
	//Analogutgång
	M AT %M*		: BOOL;		//Handställning~wp:[trendoptions]i:14400, t:1
	OPM AT %M* 		: REAL;		//Värde handställning~wp:[unit]%[format]0.0
	
	//Analogingång
	rCal 					: REAL; 	//Kalibrering
	iMedelvardeSekunder 	: UDINT := 0;
	AI_OPM					: REAL; 	//Manuellt värde~wp:
	
